REGION Network 44: E5CC[3]-Write TempSP + AlarmValue1 ~ AlarmValue2_LowerLimit Command
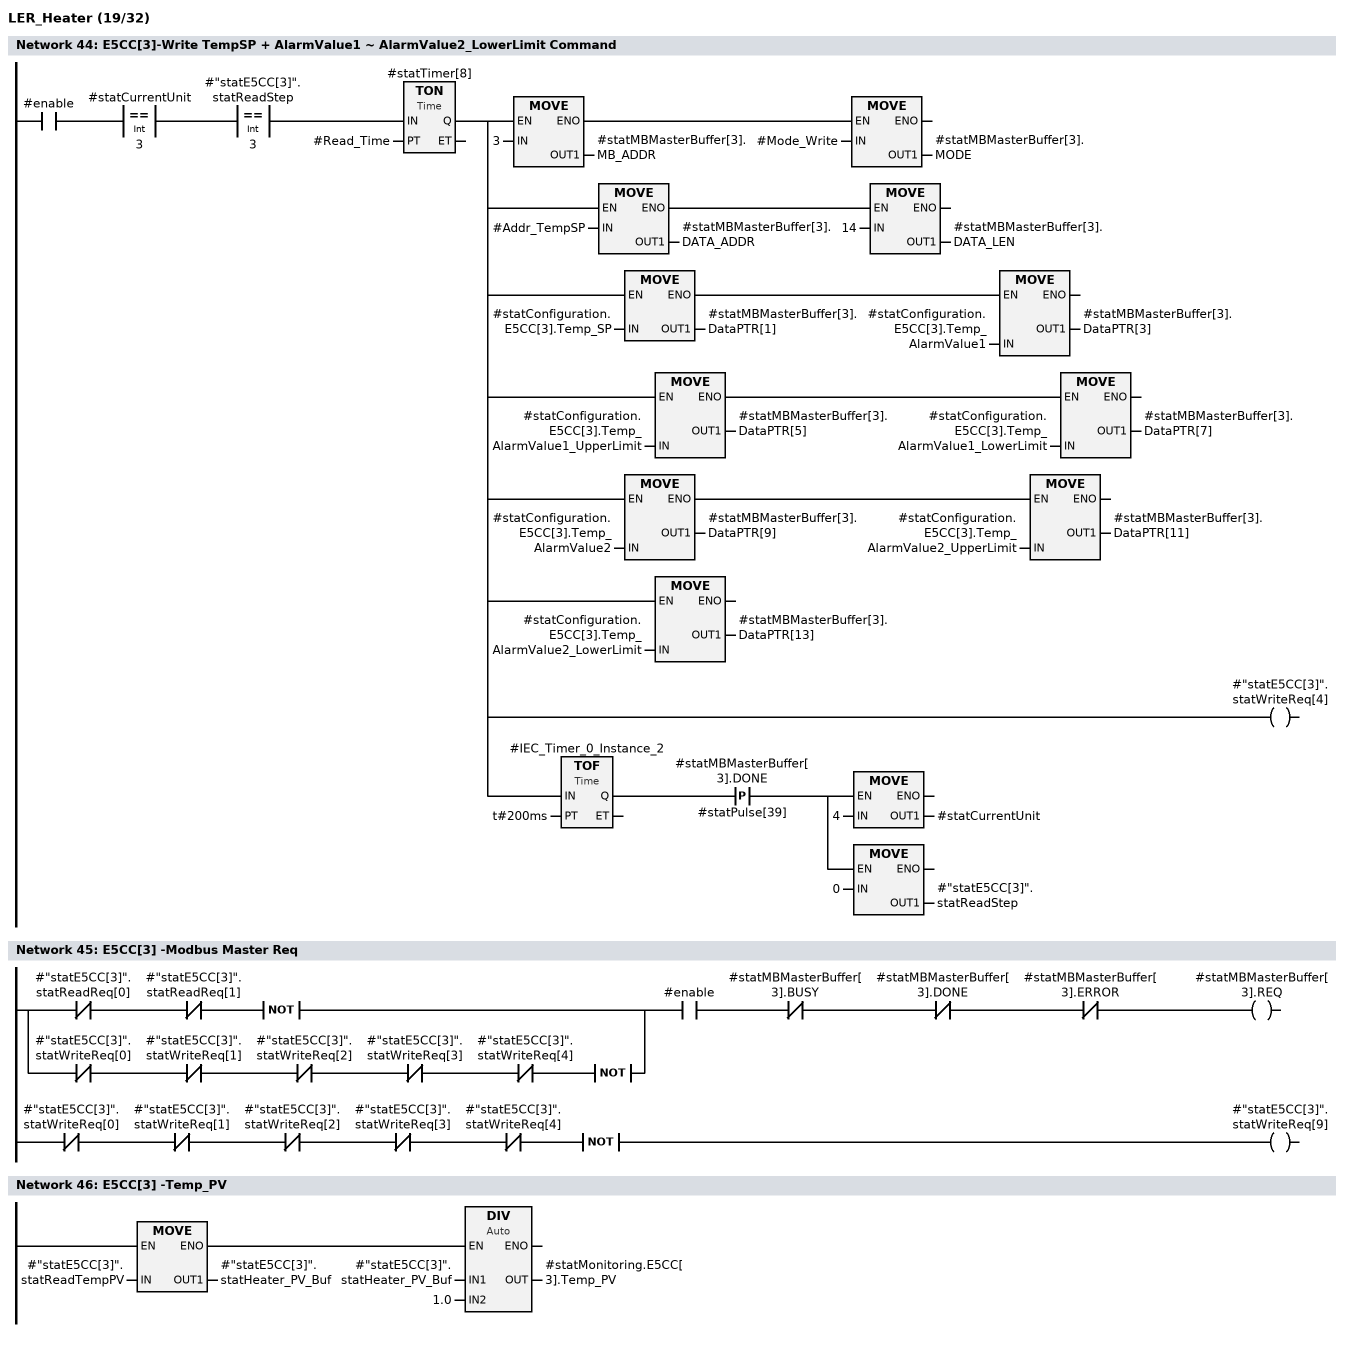
   RUNG wire#powerrail
      Contact( #enable )
      { S7_Templates := "SrcType := Int" } EQ_Contact(in1 := #statCurrentUnit, in2 := 3)
      { S7_Templates := "SrcType := Int" } EQ_Contact(in1 := #"statE5CC[3]".statReadStep, in2 := 3)
      { S7_Templates := "time_type := Time" } #statTimer[8].TON(pt := #Read_Time, et =>)
      wire#w1
      Move(in := 3, out1 => #statMBMasterBuffer[3].MB_ADDR)
      Move(in := #Mode_Write, out1 => #statMBMasterBuffer[3].MODE)
   END_RUNG
   RUNG wire#w1
      Move(in := #Addr_TempSP, out1 => #statMBMasterBuffer[3].DATA_ADDR)
      Move(in := 14, out1 => #statMBMasterBuffer[3].DATA_LEN)
   END_RUNG
   RUNG wire#w1
      Move(in := #statConfiguration.E5CC[3].Temp_SP, out1 => #statMBMasterBuffer[3].DataPTR[1])
      Move(in := #statConfiguration.E5CC[3].Temp_AlarmValue1, out1 => #statMBMasterBuffer[3].DataPTR[3])
   END_RUNG
   RUNG wire#w1
      Move(in := #statConfiguration.E5CC[3].Temp_AlarmValue1_UpperLimit, out1 => #statMBMasterBuffer[3].DataPTR[5])
      Move(in := #statConfiguration.E5CC[3].Temp_AlarmValue1_LowerLimit, out1 => #statMBMasterBuffer[3].DataPTR[7])
   END_RUNG
   RUNG wire#w1
      Move(in := #statConfiguration.E5CC[3].Temp_AlarmValue2, out1 => #statMBMasterBuffer[3].DataPTR[9])
      Move(in := #statConfiguration.E5CC[3].Temp_AlarmValue2_UpperLimit, out1 => #statMBMasterBuffer[3].DataPTR[11])
   END_RUNG
   RUNG wire#w1
      Move(in := #statConfiguration.E5CC[3].Temp_AlarmValue2_LowerLimit, out1 => #statMBMasterBuffer[3].DataPTR[13])
   END_RUNG
   RUNG wire#w1
      Coil( #"statE5CC[3]".statWriteReq[4] )
   END_RUNG
   RUNG wire#w1
      { S7_Templates := "time_type := Time" } #IEC_Timer_0_Instance_2.TOF(pt := t#200ms, et =>)
      P_Contact(operand := #statMBMasterBuffer[3].DONE, bit := #statPulse[39])
      wire#w2
      Move(in := 4, out1 => #statCurrentUnit)
   END_RUNG
   RUNG wire#w2
      Move(in := 0, out1 => #"statE5CC[3]".statReadStep)
   END_RUNG
   // the same network as SCL:
   #statTimer[8].TON(IN := #enable AND (#statCurrentUnit = 3) AND (#"statE5CC[3]".statReadStep = 3),
                     PT := #Read_Time);
   IF #statTimer[8].Q THEN
       #statMBMasterBuffer[3].MB_ADDR := 3;
       #statMBMasterBuffer[3].MODE := #Mode_Write;
       #statMBMasterBuffer[3].DATA_ADDR := #Addr_TempSP;
       #statMBMasterBuffer[3].DATA_LEN := 14;
       #statMBMasterBuffer[3].DataPTR[1] := #statConfiguration.E5CC[3].Temp_SP;
       #statMBMasterBuffer[3].DataPTR[3] := #statConfiguration.E5CC[3].Temp_AlarmValue1;
       #statMBMasterBuffer[3].DataPTR[5] := #statConfiguration.E5CC[3].Temp_AlarmValue1_UpperLimit;
       #statMBMasterBuffer[3].DataPTR[7] := #statConfiguration.E5CC[3].Temp_AlarmValue1_LowerLimit;
       #statMBMasterBuffer[3].DataPTR[9] := #statConfiguration.E5CC[3].Temp_AlarmValue2;
       #statMBMasterBuffer[3].DataPTR[11] := #statConfiguration.E5CC[3].Temp_AlarmValue2_UpperLimit;
       #statMBMasterBuffer[3].DataPTR[13] := #statConfiguration.E5CC[3].Temp_AlarmValue2_LowerLimit;
   END_IF;
   #"statE5CC[3]".statWriteReq[4] := #statTimer[8].Q;
   #IEC_Timer_0_Instance_2(IN := #statTimer[8].Q, PT := t#200ms);   // TOF
   #_w1 := #IEC_Timer_0_Instance_2.Q AND #statMBMasterBuffer[3].DONE AND NOT #statPulse[39];   // rising edge of #statMBMasterBuffer[3].DONE
   #statPulse[39] := #statMBMasterBuffer[3].DONE;
   IF #_w1 THEN
       #statCurrentUnit := 4;
       #"statE5CC[3]".statReadStep := 0;
   END_IF;
END_REGION

REGION Network 45: E5CC[3] -Modbus Master Req
   RUNG wire#powerrail
      I_Contact( #"statE5CC[3]".statReadReq[0] )
      I_Contact( #"statE5CC[3]".statReadReq[1] )
      Not()
      wire#w1
      Contact( #enable )
      I_Contact( #statMBMasterBuffer[3].BUSY )
      I_Contact( #statMBMasterBuffer[3].DONE )
      I_Contact( #statMBMasterBuffer[3].ERROR )
      Coil( #statMBMasterBuffer[3].REQ )
   END_RUNG
   RUNG wire#powerrail
      I_Contact( #"statE5CC[3]".statWriteReq[0] )
      I_Contact( #"statE5CC[3]".statWriteReq[1] )
      I_Contact( #"statE5CC[3]".statWriteReq[2] )
      I_Contact( #"statE5CC[3]".statWriteReq[3] )
      I_Contact( #"statE5CC[3]".statWriteReq[4] )
      Not()
   END_RUNG wire#w1
   RUNG wire#powerrail
      I_Contact( #"statE5CC[3]".statWriteReq[0] )
      I_Contact( #"statE5CC[3]".statWriteReq[1] )
      I_Contact( #"statE5CC[3]".statWriteReq[2] )
      I_Contact( #"statE5CC[3]".statWriteReq[3] )
      I_Contact( #"statE5CC[3]".statWriteReq[4] )
      Not()
      Coil( #"statE5CC[3]".statWriteReq[9] )
   END_RUNG
   // the same network as SCL:
   #statMBMasterBuffer[3].REQ := (NOT (NOT #"statE5CC[3]".statReadReq[0] AND NOT #"statE5CC[3]".statReadReq[1]) OR NOT (NOT #"statE5CC[3]".statWriteReq[0] AND NOT #"statE5CC[3]".statWriteReq[1] AND NOT #"statE5CC[3]".statWriteReq[2] AND NOT #"statE5CC[3]".statWriteReq[3] AND NOT #"statE5CC[3]".statWriteReq[4])) AND #enable AND NOT #statMBMasterBuffer[3].BUSY AND NOT #statMBMasterBuffer[3].DONE AND NOT #statMBMasterBuffer[3].ERROR;
   #"statE5CC[3]".statWriteReq[9] := NOT (NOT #"statE5CC[3]".statWriteReq[0] AND NOT #"statE5CC[3]".statWriteReq[1] AND NOT #"statE5CC[3]".statWriteReq[2] AND NOT #"statE5CC[3]".statWriteReq[3] AND NOT #"statE5CC[3]".statWriteReq[4]);
END_REGION

REGION Network 46: E5CC[3] -Temp_PV
   RUNG wire#powerrail
      Move(in := #"statE5CC[3]".statReadTempPV, out1 => #"statE5CC[3]".statHeater_PV_Buf)
      Div(in1 := #"statE5CC[3]".statHeater_PV_Buf, in2 := 1.0, out => #statMonitoring.E5CC[3].Temp_PV)
   END_RUNG
   // the same network as SCL:
   #"statE5CC[3]".statHeater_PV_Buf := #"statE5CC[3]".statReadTempPV;
   #statMonitoring.E5CC[3].Temp_PV := #"statE5CC[3]".statHeater_PV_Buf / 1.0;
END_REGION

REGION Network 47: E5CC[3] -Temp_PV Complete Check
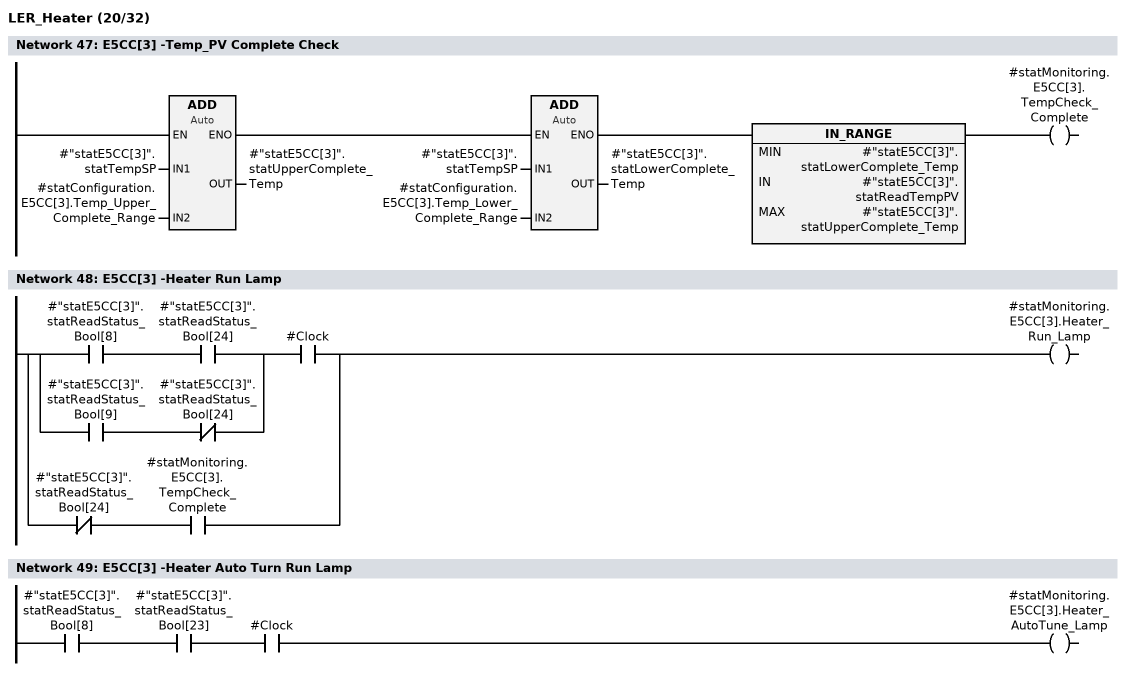
   RUNG wire#powerrail
      Add(in1 := #"statE5CC[3]".statTempSP, in2 := #statConfiguration.E5CC[3].Temp_Upper_Complete_Range, out => #"statE5CC[3]".statUpperComplete_Temp)
      Add(in1 := #"statE5CC[3]".statTempSP, in2 := #statConfiguration.E5CC[3].Temp_Lower_Complete_Range, out => #"statE5CC[3]".statLowerComplete_Temp)
      { S7_Templates := "SrcType := Real" } InRange(min := #"statE5CC[3]".statLowerComplete_Temp, in := #"statE5CC[3]".statReadTempPV, max := #"statE5CC[3]".statUpperComplete_Temp)
      Coil( #statMonitoring.E5CC[3].TempCheck_Complete )
   END_RUNG
   // the same network as SCL:
   #"statE5CC[3]".statUpperComplete_Temp := #"statE5CC[3]".statTempSP + #statConfiguration.E5CC[3].Temp_Upper_Complete_Range;
   #"statE5CC[3]".statLowerComplete_Temp := #"statE5CC[3]".statTempSP + #statConfiguration.E5CC[3].Temp_Lower_Complete_Range;
   #statMonitoring.E5CC[3].TempCheck_Complete := (#"statE5CC[3]".statLowerComplete_Temp <= #"statE5CC[3]".statReadTempPV) AND (#"statE5CC[3]".statReadTempPV <= #"statE5CC[3]".statUpperComplete_Temp);
END_REGION

REGION Network 48: E5CC[3] -Heater Run Lamp
   RUNG wire#powerrail
      Contact( #"statE5CC[3]".statReadStatus_Bool[8] )
      Contact( #"statE5CC[3]".statReadStatus_Bool[24] )
      wire#w1
      Contact( #Clock )
      wire#w2
      Coil( #statMonitoring.E5CC[3].Heater_Run_Lamp )
   END_RUNG
   RUNG wire#powerrail
      Contact( #"statE5CC[3]".statReadStatus_Bool[9] )
      I_Contact( #"statE5CC[3]".statReadStatus_Bool[24] )
   END_RUNG wire#w1
   RUNG wire#powerrail
      I_Contact( #"statE5CC[3]".statReadStatus_Bool[24] )
      Contact( #statMonitoring.E5CC[3].TempCheck_Complete )
   END_RUNG wire#w2
   // the same network as SCL:
   #statMonitoring.E5CC[3].Heater_Run_Lamp := (((#"statE5CC[3]".statReadStatus_Bool[8] AND #"statE5CC[3]".statReadStatus_Bool[24]) OR (#"statE5CC[3]".statReadStatus_Bool[9] AND NOT #"statE5CC[3]".statReadStatus_Bool[24])) AND #Clock) OR (NOT #"statE5CC[3]".statReadStatus_Bool[24] AND #statMonitoring.E5CC[3].TempCheck_Complete);
END_REGION

REGION Network 49: E5CC[3] -Heater Auto Turn Run Lamp
   RUNG wire#powerrail
      Contact( #"statE5CC[3]".statReadStatus_Bool[8] )
      Contact( #"statE5CC[3]".statReadStatus_Bool[23] )
      Contact( #Clock )
      Coil( #statMonitoring.E5CC[3].Heater_AutoTune_Lamp )
   END_RUNG
   // the same network as SCL:
   #statMonitoring.E5CC[3].Heater_AutoTune_Lamp := #"statE5CC[3]".statReadStatus_Bool[8] AND #"statE5CC[3]".statReadStatus_Bool[23] AND #Clock;
END_REGION

REGION Network 50 (SCL): E5CC[3] -Error Check
   REGION  E5CC Error Status
       // Dword to Bool
       SCATTER(IN := #"statE5CC[3]".statReadStatus,
               OUT => #"statE5CC[3]".statReadStatus_Bool);
   END_REGION


   REGION Error Code Search
       IF #"statE5CC[3]".statReadStatus <> 0 THEN
           CASE #"statE5CC[3]".statReadStatus OF
               #ERR_HEATER_CURRENT_VALUE_EXCEEDED_CT1:
                   #statMonitoring.E5CC[3].Status := #ERR_HEATER_CURRENT_VALUE_EXCEEDED_CT1;
               #ERR_HEATER_CURRENT_VALUE_HOLD_CT1:
                   #statMonitoring.E5CC[3].Status := #ERR_HEATER_CURRENT_VALUE_HOLD_CT1;
               #ERR_AD_CONVERTER_ABNORMALITY:
                   #statMonitoring.E5CC[3].Status := #ERR_AD_CONVERTER_ABNORMALITY;
               #ERR_HS_SSR_FAULT_ALERT_CT1:
                   #statMonitoring.E5CC[3].Status := #ERR_HS_SSR_FAULT_ALERT_CT1;
               #ERR_RSP_INPUT_ABNORMALITIES:
                   #statMonitoring.E5CC[3].Status := #ERR_RSP_INPUT_ABNORMALITIES;
               #ERR_MORE_THAN_INPUT:
                   #statMonitoring.E5CC[3].Status := #ERR_MORE_THAN_INPUT;
               #ERR_POTENTIOMETER_INPUT_ABNORMAL:
                   #statMonitoring.E5CC[3].Status := #ERR_POTENTIOMETER_INPUT_ABNORMAL;
               #ERR_CONTROL_OUTPUT_HEATED_OPEN_OUTPUT:
                   #statMonitoring.E5CC[3].Status := #ERR_CONTROL_OUTPUT_HEATED_OPEN_OUTPUT;
               #ERR_CONTROL_OUTPUT_COOL_CLOSE_OUTPUT:
                   #statMonitoring.E5CC[3].Status := #ERR_CONTROL_OUTPUT_COOL_CLOSE_OUTPUT;
               #ERR_HEATER_OPEN_CIRCUIT_HB_ALARM_CT1:
                   #statMonitoring.E5CC[3].Status := #ERR_HEATER_OPEN_CIRCUIT_HB_ALARM_CT1;
               #ERR_HEATER_OPEN_CIRCUIT_HB_ALARM_CT2:
                   #statMonitoring.E5CC[3].Status := #ERR_HEATER_OPEN_CIRCUIT_HB_ALARM_CT2;
               #ERR_ALERT_1:
                   #statMonitoring.E5CC[3].Status := #ERR_ALERT_1;
               #ERR_ALERT_2:
                   #statMonitoring.E5CC[3].Status := #ERR_ALERT_2;
               #ERR_ALERT_3:
                   #statMonitoring.E5CC[3].Status := #ERR_ALERT_3;
               #ERR_PROGRAM_END_OUTPUT:
                   #statMonitoring.E5CC[3].Status := #ERR_PROGRAM_END_OUTPUT;
               #ERR_EVENT_INPUT_1:
                   #statMonitoring.E5CC[3].Status := #ERR_EVENT_INPUT_1;
               #ERR_EVENT_INPUT_2:
                   #statMonitoring.E5CC[3].Status := #ERR_EVENT_INPUT_2;
               #ERR_EVENT_INPUT_3:
                   #statMonitoring.E5CC[3].Status := #ERR_EVENT_INPUT_3;
               #ERR_EVENT_INPUT_4:
                   #statMonitoring.E5CC[3].Status := #ERR_EVENT_INPUT_4;
               #ERR_WRITE_MODE:
                   #statMonitoring.E5CC[3].Status := #ERR_WRITE_MODE;
               #ERR_NON_VOLATILE_MEMORY:
                   #statMonitoring.E5CC[3].Status := #ERR_NON_VOLATILE_MEMORY;
               #ERR_SETTING_AREA:
                   #statMonitoring.E5CC[3].Status := #ERR_SETTING_AREA;
               #ERR_AT_RUN_STOP:
                   #statMonitoring.E5CC[3].Status := #ERR_AT_RUN_STOP;
               #ERR_RUN_STOP:
                   #statMonitoring.E5CC[3].Status := #ERR_RUN_STOP;
               #ERR_COMMUNICATION_WRITE:
                   #statMonitoring.E5CC[3].Status := #ERR_COMMUNICATION_WRITE;
               #ERR_AUTO_MANUAL:
                   #statMonitoring.E5CC[3].Status := #ERR_AUTO_MANUAL;
               #ERR_PROGRAM_START:
                   #statMonitoring.E5CC[3].Status := #ERR_PROGRAM_START;
               #ERR_HEATER_CURRENT_VALUE_EXCEEDED_CT2:
                   #statMonitoring.E5CC[3].Status := #ERR_HEATER_CURRENT_VALUE_EXCEEDED_CT2;
               #ERR_HEATER_CURRENT_VALUE_HOLD_CT2:
                   #statMonitoring.E5CC[3].Status := #ERR_HEATER_CURRENT_VALUE_HOLD_CT2;
               #ERR_HS_SSR_FAILURE_ALARM_CT2:
                   #statMonitoring.E5CC[3].Status := #ERR_HS_SSR_FAILURE_ALARM_CT2;
           END_CASE;
       ELSIF #"statE5CC[3]".statReadStatus = 0 THEN
           #statMonitoring.E5CC[3].Status := 0;
       END_IF;
   END_REGION

   #statMonitoring.E5CC[3].Error := #"statE5CC[3]".statReadStatus <> 0;
END_REGION

REGION Network 51 (SCL): E5CC[3]-##### Outputs mapping #####
   // Output Mapping
   #statMonitoring.E5CC[3].Temp_SP := #"statE5CC[3]".statTempSP;
   #statMonitoring.E5CC[3].Temp_AlarmValue1 := #"statE5CC[3]".statAlarmValue1;
   #statMonitoring.E5CC[3].Temp_AlarmValue1_UpperLimit := #"statE5CC[3]".statAlarmValue1_UpperLimit;
   #statMonitoring.E5CC[3].Temp_AlarmValue1_LowerLimit := #"statE5CC[3]".statAlarmValue1_LowerLimit;
   #statMonitoring.E5CC[3].Temp_AlarmValue2 := #"statE5CC[3]".statAlarmValue2;
   #statMonitoring.E5CC[3].Temp_AlarmValue2_UpperLimit := #"statE5CC[3]".statAlarmValue2_UpperLimit;
   #statMonitoring.E5CC[3].Temp_AlarmValue2_LowerLimit := #"statE5CC[3]".statAlarmValue2_LowerLimit;
   #statMonitoring.E5CC[3].E5CC_Status := #"statE5CC[3]".statReadStatus;
   #statMonitoring.E5CC[3].E5CC_Status_Bool := #"statE5CC[3]".statReadStatus_Bool;
END_REGION

REGION Network 52: E5CC[4] - ###### Input Mapping ######
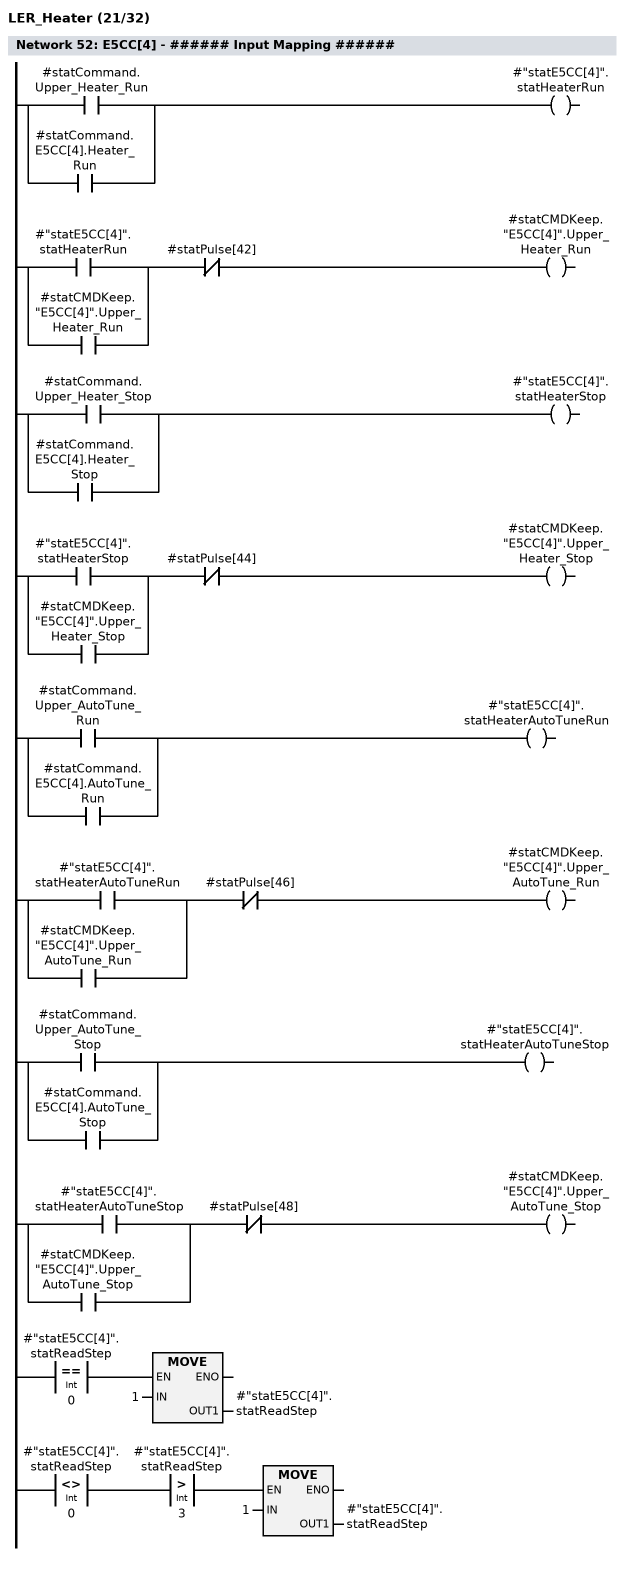
   RUNG wire#powerrail
      Contact( #statCommand.Upper_Heater_Run )
      wire#w1
      Coil( #"statE5CC[4]".statHeaterRun )
   END_RUNG
   RUNG wire#powerrail
      Contact( #statCommand.E5CC[4].Heater_Run )
   END_RUNG wire#w1
   RUNG wire#powerrail
      Contact( #"statE5CC[4]".statHeaterRun )
      wire#w2
      I_Contact( #statPulse[42] )
      Coil( #statCMDKeep."E5CC[4]".Upper_Heater_Run )
   END_RUNG
   RUNG wire#powerrail
      Contact( #statCMDKeep."E5CC[4]".Upper_Heater_Run )
   END_RUNG wire#w2
   RUNG wire#powerrail
      Contact( #statCommand.Upper_Heater_Stop )
      wire#w3
      Coil( #"statE5CC[4]".statHeaterStop )
   END_RUNG
   RUNG wire#powerrail
      Contact( #statCommand.E5CC[4].Heater_Stop )
   END_RUNG wire#w3
   RUNG wire#powerrail
      Contact( #"statE5CC[4]".statHeaterStop )
      wire#w4
      I_Contact( #statPulse[44] )
      Coil( #statCMDKeep."E5CC[4]".Upper_Heater_Stop )
   END_RUNG
   RUNG wire#powerrail
      Contact( #statCMDKeep."E5CC[4]".Upper_Heater_Stop )
   END_RUNG wire#w4
   RUNG wire#powerrail
      Contact( #statCommand.Upper_AutoTune_Run )
      wire#w5
      Coil( #"statE5CC[4]".statHeaterAutoTuneRun )
   END_RUNG
   RUNG wire#powerrail
      Contact( #statCommand.E5CC[4].AutoTune_Run )
   END_RUNG wire#w5
   RUNG wire#powerrail
      Contact( #"statE5CC[4]".statHeaterAutoTuneRun )
      wire#w6
      I_Contact( #statPulse[46] )
      Coil( #statCMDKeep."E5CC[4]".Upper_AutoTune_Run )
   END_RUNG
   RUNG wire#powerrail
      Contact( #statCMDKeep."E5CC[4]".Upper_AutoTune_Run )
   END_RUNG wire#w6
   RUNG wire#powerrail
      Contact( #statCommand.Upper_AutoTune_Stop )
      wire#w7
      Coil( #"statE5CC[4]".statHeaterAutoTuneStop )
   END_RUNG
   RUNG wire#powerrail
      Contact( #statCommand.E5CC[4].AutoTune_Stop )
   END_RUNG wire#w7
   RUNG wire#powerrail
      Contact( #"statE5CC[4]".statHeaterAutoTuneStop )
      wire#w8
      I_Contact( #statPulse[48] )
      Coil( #statCMDKeep."E5CC[4]".Upper_AutoTune_Stop )
   END_RUNG
   RUNG wire#powerrail
      Contact( #statCMDKeep."E5CC[4]".Upper_AutoTune_Stop )
   END_RUNG wire#w8
   RUNG wire#powerrail
      { S7_Templates := "SrcType := Int" } EQ_Contact(in1 := #"statE5CC[4]".statReadStep, in2 := 0)
      Move(in := 1, out1 => #"statE5CC[4]".statReadStep)
   END_RUNG
   RUNG wire#powerrail
      { S7_Templates := "SrcType := Int" } NE_Contact(in1 := #"statE5CC[4]".statReadStep, in2 := 0)
      { S7_Templates := "SrcType := Int" } GT_Contact(in1 := #"statE5CC[4]".statReadStep, in2 := 3)
      Move(in := 1, out1 => #"statE5CC[4]".statReadStep)
   END_RUNG
   // the same network as SCL:
   #"statE5CC[4]".statHeaterRun := #statCommand.Upper_Heater_Run OR #statCommand.E5CC[4].Heater_Run;
   #statCMDKeep."E5CC[4]".Upper_Heater_Run := (#"statE5CC[4]".statHeaterRun OR #statCMDKeep."E5CC[4]".Upper_Heater_Run) AND NOT #statPulse[42];
   #"statE5CC[4]".statHeaterStop := #statCommand.Upper_Heater_Stop OR #statCommand.E5CC[4].Heater_Stop;
   #statCMDKeep."E5CC[4]".Upper_Heater_Stop := (#"statE5CC[4]".statHeaterStop OR #statCMDKeep."E5CC[4]".Upper_Heater_Stop) AND NOT #statPulse[44];
   #"statE5CC[4]".statHeaterAutoTuneRun := #statCommand.Upper_AutoTune_Run OR #statCommand.E5CC[4].AutoTune_Run;
   #statCMDKeep."E5CC[4]".Upper_AutoTune_Run := (#"statE5CC[4]".statHeaterAutoTuneRun OR #statCMDKeep."E5CC[4]".Upper_AutoTune_Run) AND NOT #statPulse[46];
   #"statE5CC[4]".statHeaterAutoTuneStop := #statCommand.Upper_AutoTune_Stop OR #statCommand.E5CC[4].AutoTune_Stop;
   #statCMDKeep."E5CC[4]".Upper_AutoTune_Stop := (#"statE5CC[4]".statHeaterAutoTuneStop OR #statCMDKeep."E5CC[4]".Upper_AutoTune_Stop) AND NOT #statPulse[48];
   IF #"statE5CC[4]".statReadStep = 0 THEN #"statE5CC[4]".statReadStep := 1; END_IF;
   IF (#"statE5CC[4]".statReadStep <> 0) AND (#"statE5CC[4]".statReadStep > 3) THEN
       #"statE5CC[4]".statReadStep := 1;
   END_IF;
END_REGION

REGION Network 53: E5CC[4] -Read Temp PV + Status Command
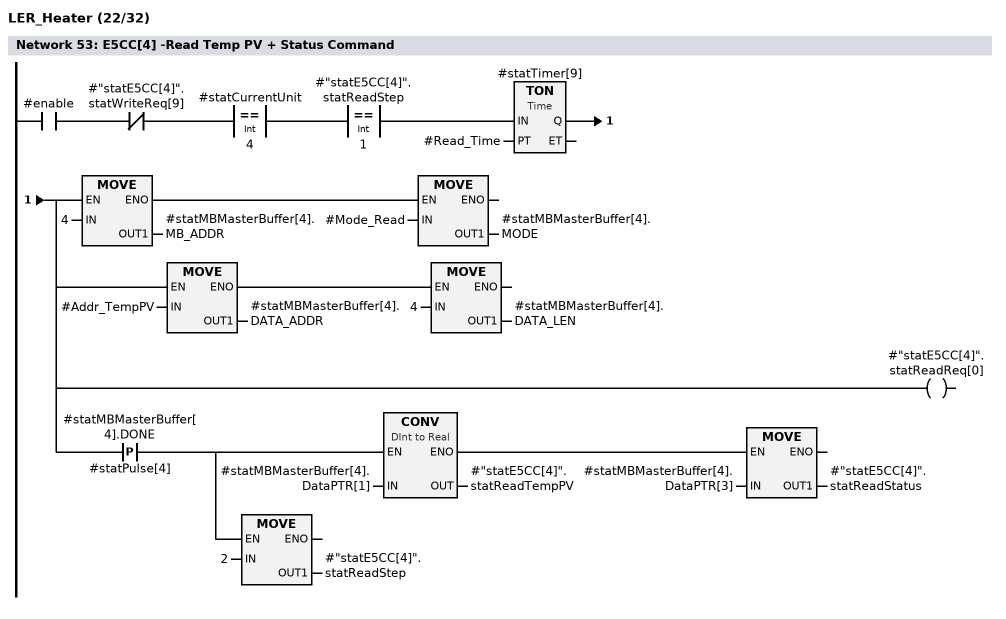
   RUNG wire#powerrail
      Contact( #enable )
      I_Contact( #"statE5CC[4]".statWriteReq[9] )
      { S7_Templates := "SrcType := Int" } EQ_Contact(in1 := #statCurrentUnit, in2 := 4)
      { S7_Templates := "SrcType := Int" } EQ_Contact(in1 := #"statE5CC[4]".statReadStep, in2 := 1)
      { S7_Templates := "time_type := Time" } #statTimer[9].TON(pt := #Read_Time, et =>)
      wire#w1
      Move(in := 4, out1 => #statMBMasterBuffer[4].MB_ADDR)
      Move(in := #Mode_Read, out1 => #statMBMasterBuffer[4].MODE)
   END_RUNG
   RUNG wire#w1
      Move(in := #Addr_TempPV, out1 => #statMBMasterBuffer[4].DATA_ADDR)
      Move(in := 4, out1 => #statMBMasterBuffer[4].DATA_LEN)
   END_RUNG
   RUNG wire#w1
      Coil( #"statE5CC[4]".statReadReq[0] )
   END_RUNG
   RUNG wire#w1
      P_Contact(operand := #statMBMasterBuffer[4].DONE, bit := #statPulse[4])
      wire#w2
      { S7_Templates := "[SrcType := DInt, DestType := Real]" } Convert(in := #statMBMasterBuffer[4].DataPTR[1], out => #"statE5CC[4]".statReadTempPV)
      Move(in := #statMBMasterBuffer[4].DataPTR[3], out1 => #"statE5CC[4]".statReadStatus)
   END_RUNG
   RUNG wire#w2
      Move(in := 2, out1 => #"statE5CC[4]".statReadStep)
   END_RUNG
   // the same network as SCL:
   #statTimer[9].TON(IN := #enable AND NOT #"statE5CC[4]".statWriteReq[9] AND (#statCurrentUnit = 4) AND (#"statE5CC[4]".statReadStep = 1),
                     PT := #Read_Time);
   IF #statTimer[9].Q THEN
       #statMBMasterBuffer[4].MB_ADDR := 4;
       #statMBMasterBuffer[4].MODE := #Mode_Read;
       #statMBMasterBuffer[4].DATA_ADDR := #Addr_TempPV;
       #statMBMasterBuffer[4].DATA_LEN := 4;
   END_IF;
   #"statE5CC[4]".statReadReq[0] := #statTimer[9].Q;
   #_w1 := #statTimer[9].Q AND #statMBMasterBuffer[4].DONE AND NOT #statPulse[4];   // rising edge of #statMBMasterBuffer[4].DONE
   #statPulse[4] := #statMBMasterBuffer[4].DONE;
   IF #_w1 THEN
       #"statE5CC[4]".statReadTempPV := DINT_TO_REAL(#statMBMasterBuffer[4].DataPTR[1]);
       #"statE5CC[4]".statReadStatus := #statMBMasterBuffer[4].DataPTR[3];
       #"statE5CC[4]".statReadStep := 2;
   END_IF;
END_REGION

REGION Network 54: E5CC[4] -Read TempSP + AlarmValue1 ~ AlarmValue2_LowerLimit Commad
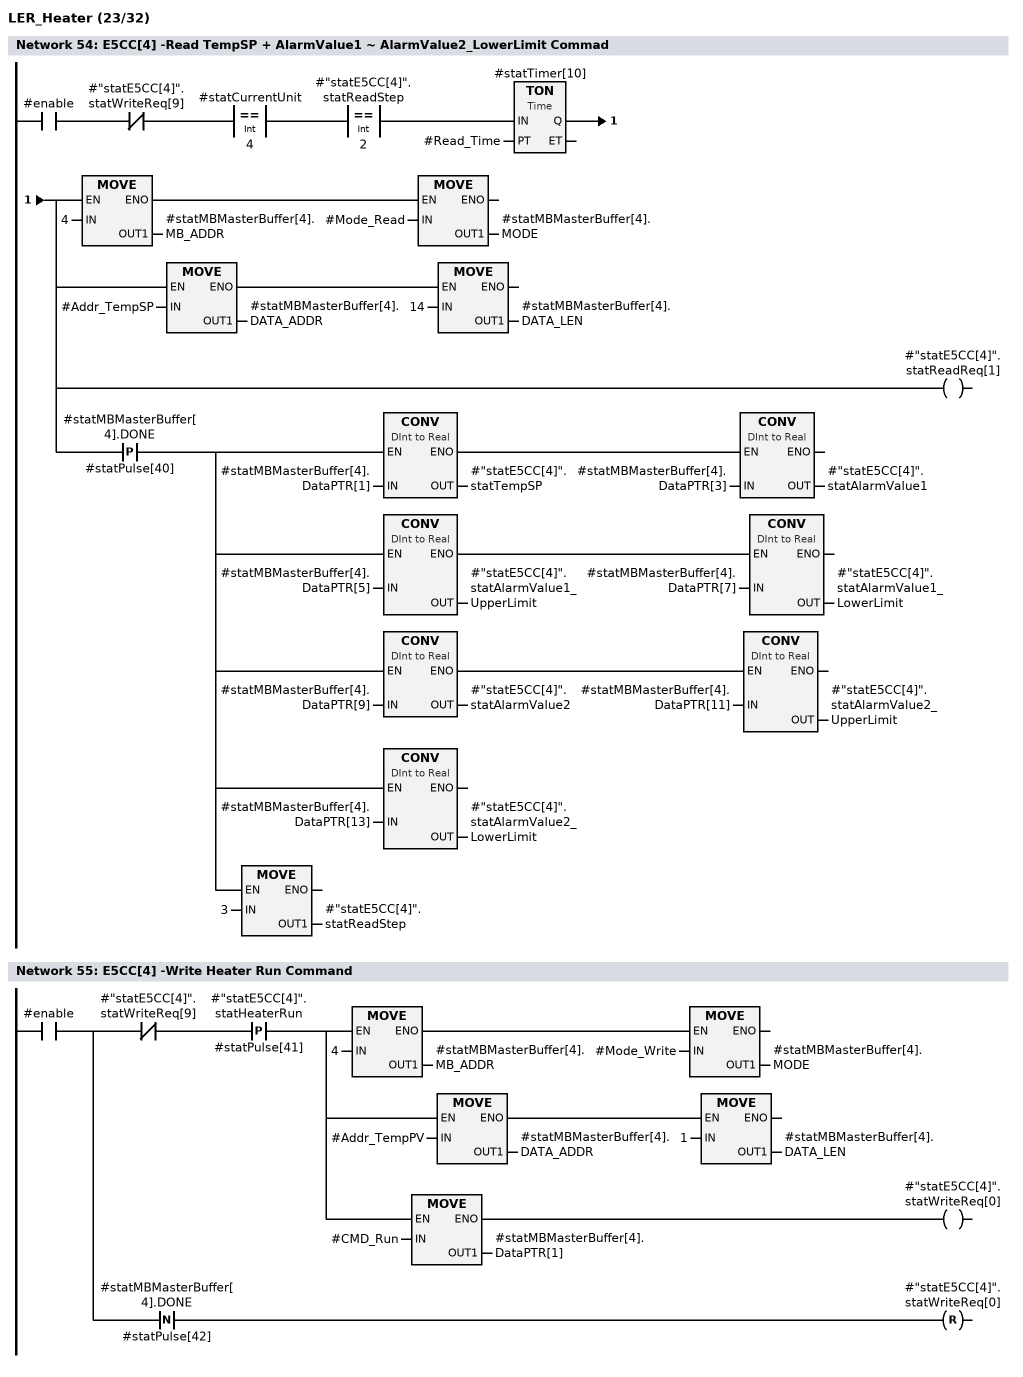
   RUNG wire#powerrail
      Contact( #enable )
      I_Contact( #"statE5CC[4]".statWriteReq[9] )
      { S7_Templates := "SrcType := Int" } EQ_Contact(in1 := #statCurrentUnit, in2 := 4)
      { S7_Templates := "SrcType := Int" } EQ_Contact(in1 := #"statE5CC[4]".statReadStep, in2 := 2)
      { S7_Templates := "time_type := Time" } #statTimer[10].TON(pt := #Read_Time, et =>)
      wire#w1
      Move(in := 4, out1 => #statMBMasterBuffer[4].MB_ADDR)
      Move(in := #Mode_Read, out1 => #statMBMasterBuffer[4].MODE)
   END_RUNG
   RUNG wire#w1
      Move(in := #Addr_TempSP, out1 => #statMBMasterBuffer[4].DATA_ADDR)
      Move(in := 14, out1 => #statMBMasterBuffer[4].DATA_LEN)
   END_RUNG
   RUNG wire#w1
      Coil( #"statE5CC[4]".statReadReq[1] )
   END_RUNG
   RUNG wire#w1
      P_Contact(operand := #statMBMasterBuffer[4].DONE, bit := #statPulse[40])
      wire#w2
      { S7_Templates := "[SrcType := DInt, DestType := Real]" } Convert(in := #statMBMasterBuffer[4].DataPTR[1], out => #"statE5CC[4]".statTempSP)
      { S7_Templates := "[SrcType := DInt, DestType := Real]" } Convert(in := #statMBMasterBuffer[4].DataPTR[3], out => #"statE5CC[4]".statAlarmValue1)
   END_RUNG
   RUNG wire#w2
      { S7_Templates := "[SrcType := DInt, DestType := Real]" } Convert(in := #statMBMasterBuffer[4].DataPTR[5], out => #"statE5CC[4]".statAlarmValue1_UpperLimit)
      { S7_Templates := "[SrcType := DInt, DestType := Real]" } Convert(in := #statMBMasterBuffer[4].DataPTR[7], out => #"statE5CC[4]".statAlarmValue1_LowerLimit)
   END_RUNG
   RUNG wire#w2
      { S7_Templates := "[SrcType := DInt, DestType := Real]" } Convert(in := #statMBMasterBuffer[4].DataPTR[9], out => #"statE5CC[4]".statAlarmValue2)
      { S7_Templates := "[SrcType := DInt, DestType := Real]" } Convert(in := #statMBMasterBuffer[4].DataPTR[11], out => #"statE5CC[4]".statAlarmValue2_UpperLimit)
   END_RUNG
   RUNG wire#w2
      { S7_Templates := "[SrcType := DInt, DestType := Real]" } Convert(in := #statMBMasterBuffer[4].DataPTR[13], out => #"statE5CC[4]".statAlarmValue2_LowerLimit)
   END_RUNG
   RUNG wire#w2
      Move(in := 3, out1 => #"statE5CC[4]".statReadStep)
   END_RUNG
   // the same network as SCL:
   #statTimer[10].TON(IN := #enable AND NOT #"statE5CC[4]".statWriteReq[9] AND (#statCurrentUnit = 4) AND (#"statE5CC[4]".statReadStep = 2),
                      PT := #Read_Time);
   IF #statTimer[10].Q THEN
       #statMBMasterBuffer[4].MB_ADDR := 4;
       #statMBMasterBuffer[4].MODE := #Mode_Read;
       #statMBMasterBuffer[4].DATA_ADDR := #Addr_TempSP;
       #statMBMasterBuffer[4].DATA_LEN := 14;
   END_IF;
   #"statE5CC[4]".statReadReq[1] := #statTimer[10].Q;
   #_w1 := #statTimer[10].Q AND #statMBMasterBuffer[4].DONE AND NOT #statPulse[40];   // rising edge of #statMBMasterBuffer[4].DONE
   #statPulse[40] := #statMBMasterBuffer[4].DONE;
   IF #_w1 THEN
       #"statE5CC[4]".statTempSP := DINT_TO_REAL(#statMBMasterBuffer[4].DataPTR[1]);
       #"statE5CC[4]".statAlarmValue1 := DINT_TO_REAL(#statMBMasterBuffer[4].DataPTR[3]);
       #"statE5CC[4]".statAlarmValue1_UpperLimit := DINT_TO_REAL(#statMBMasterBuffer[4].DataPTR[5]);
       #"statE5CC[4]".statAlarmValue1_LowerLimit := DINT_TO_REAL(#statMBMasterBuffer[4].DataPTR[7]);
       #"statE5CC[4]".statAlarmValue2 := DINT_TO_REAL(#statMBMasterBuffer[4].DataPTR[9]);
       #"statE5CC[4]".statAlarmValue2_UpperLimit := DINT_TO_REAL(#statMBMasterBuffer[4].DataPTR[11]);
       #"statE5CC[4]".statAlarmValue2_LowerLimit := DINT_TO_REAL(#statMBMasterBuffer[4].DataPTR[13]);
       #"statE5CC[4]".statReadStep := 3;
   END_IF;
END_REGION

REGION Network 55: E5CC[4] -Write Heater Run Command
   RUNG wire#powerrail
      Contact( #enable )
      wire#w1
      I_Contact( #"statE5CC[4]".statWriteReq[9] )
      P_Contact(operand := #"statE5CC[4]".statHeaterRun, bit := #statPulse[41])
      wire#w2
      Move(in := 4, out1 => #statMBMasterBuffer[4].MB_ADDR)
      Move(in := #Mode_Write, out1 => #statMBMasterBuffer[4].MODE)
   END_RUNG
   RUNG wire#w2
      Move(in := #Addr_TempPV, out1 => #statMBMasterBuffer[4].DATA_ADDR)
      Move(in := 1, out1 => #statMBMasterBuffer[4].DATA_LEN)
   END_RUNG
   RUNG wire#w2
      Move(in := #CMD_Run, out1 => #statMBMasterBuffer[4].DataPTR[1])
      Coil( #"statE5CC[4]".statWriteReq[0] )
   END_RUNG
   RUNG wire#w1
      N_Contact(operand := #statMBMasterBuffer[4].DONE, bit := #statPulse[42])
      R_Coil( #"statE5CC[4]".statWriteReq[0] )
   END_RUNG
   // the same network as SCL:
   #_w1 := #enable AND NOT #"statE5CC[4]".statWriteReq[9] AND #"statE5CC[4]".statHeaterRun AND NOT #statPulse[41];   // rising edge of #"statE5CC[4]".statHeaterRun
   #statPulse[41] := #"statE5CC[4]".statHeaterRun;
   IF #_w1 THEN
       #statMBMasterBuffer[4].MB_ADDR := 4;
       #statMBMasterBuffer[4].MODE := #Mode_Write;
       #statMBMasterBuffer[4].DATA_ADDR := #Addr_TempPV;
       #statMBMasterBuffer[4].DATA_LEN := 1;
       #statMBMasterBuffer[4].DataPTR[1] := #CMD_Run;
   END_IF;
   #"statE5CC[4]".statWriteReq[0] := #_w1;
   #_w2 := #enable AND NOT #statMBMasterBuffer[4].DONE AND #statPulse[42];   // falling edge of #statMBMasterBuffer[4].DONE
   #statPulse[42] := #statMBMasterBuffer[4].DONE;
   IF #_w2 THEN #"statE5CC[4]".statWriteReq[0] := FALSE; END_IF;
END_REGION

REGION Network 56: E5CC[4] -Write Heater Stop Command
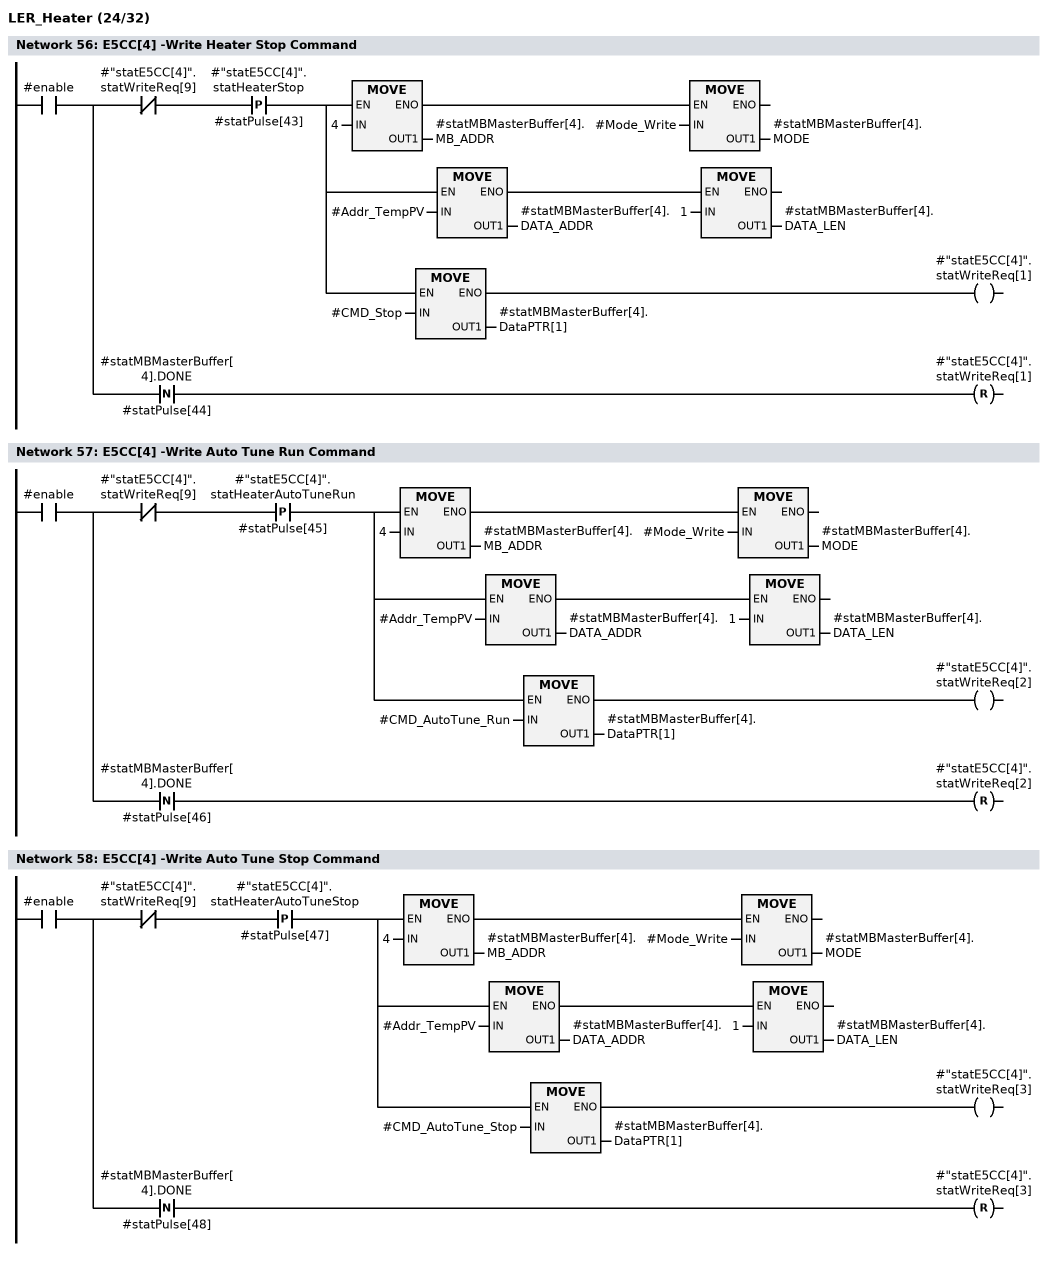
   RUNG wire#powerrail
      Contact( #enable )
      wire#w1
      I_Contact( #"statE5CC[4]".statWriteReq[9] )
      P_Contact(operand := #"statE5CC[4]".statHeaterStop, bit := #statPulse[43])
      wire#w2
      Move(in := 4, out1 => #statMBMasterBuffer[4].MB_ADDR)
      Move(in := #Mode_Write, out1 => #statMBMasterBuffer[4].MODE)
   END_RUNG
   RUNG wire#w2
      Move(in := #Addr_TempPV, out1 => #statMBMasterBuffer[4].DATA_ADDR)
      Move(in := 1, out1 => #statMBMasterBuffer[4].DATA_LEN)
   END_RUNG
   RUNG wire#w2
      Move(in := #CMD_Stop, out1 => #statMBMasterBuffer[4].DataPTR[1])
      Coil( #"statE5CC[4]".statWriteReq[1] )
   END_RUNG
   RUNG wire#w1
      N_Contact(operand := #statMBMasterBuffer[4].DONE, bit := #statPulse[44])
      R_Coil( #"statE5CC[4]".statWriteReq[1] )
   END_RUNG
   // the same network as SCL:
   #_w1 := #enable AND NOT #"statE5CC[4]".statWriteReq[9] AND #"statE5CC[4]".statHeaterStop AND NOT #statPulse[43];   // rising edge of #"statE5CC[4]".statHeaterStop
   #statPulse[43] := #"statE5CC[4]".statHeaterStop;
   IF #_w1 THEN
       #statMBMasterBuffer[4].MB_ADDR := 4;
       #statMBMasterBuffer[4].MODE := #Mode_Write;
       #statMBMasterBuffer[4].DATA_ADDR := #Addr_TempPV;
       #statMBMasterBuffer[4].DATA_LEN := 1;
       #statMBMasterBuffer[4].DataPTR[1] := #CMD_Stop;
   END_IF;
   #"statE5CC[4]".statWriteReq[1] := #_w1;
   #_w2 := #enable AND NOT #statMBMasterBuffer[4].DONE AND #statPulse[44];   // falling edge of #statMBMasterBuffer[4].DONE
   #statPulse[44] := #statMBMasterBuffer[4].DONE;
   IF #_w2 THEN #"statE5CC[4]".statWriteReq[1] := FALSE; END_IF;
END_REGION

REGION Network 57: E5CC[4] -Write Auto Tune Run Command
   RUNG wire#powerrail
      Contact( #enable )
      wire#w1
      I_Contact( #"statE5CC[4]".statWriteReq[9] )
      P_Contact(operand := #"statE5CC[4]".statHeaterAutoTuneRun, bit := #statPulse[45])
      wire#w2
      Move(in := 4, out1 => #statMBMasterBuffer[4].MB_ADDR)
      Move(in := #Mode_Write, out1 => #statMBMasterBuffer[4].MODE)
   END_RUNG
   RUNG wire#w2
      Move(in := #Addr_TempPV, out1 => #statMBMasterBuffer[4].DATA_ADDR)
      Move(in := 1, out1 => #statMBMasterBuffer[4].DATA_LEN)
   END_RUNG
   RUNG wire#w2
      Move(in := #CMD_AutoTune_Run, out1 => #statMBMasterBuffer[4].DataPTR[1])
      Coil( #"statE5CC[4]".statWriteReq[2] )
   END_RUNG
   RUNG wire#w1
      N_Contact(operand := #statMBMasterBuffer[4].DONE, bit := #statPulse[46])
      R_Coil( #"statE5CC[4]".statWriteReq[2] )
   END_RUNG
   // the same network as SCL:
   #_w1 := #enable AND NOT #"statE5CC[4]".statWriteReq[9] AND #"statE5CC[4]".statHeaterAutoTuneRun AND NOT #statPulse[45];   // rising edge of #"statE5CC[4]".statHeaterAutoTuneRun
   #statPulse[45] := #"statE5CC[4]".statHeaterAutoTuneRun;
   IF #_w1 THEN
       #statMBMasterBuffer[4].MB_ADDR := 4;
       #statMBMasterBuffer[4].MODE := #Mode_Write;
       #statMBMasterBuffer[4].DATA_ADDR := #Addr_TempPV;
       #statMBMasterBuffer[4].DATA_LEN := 1;
       #statMBMasterBuffer[4].DataPTR[1] := #CMD_AutoTune_Run;
   END_IF;
   #"statE5CC[4]".statWriteReq[2] := #_w1;
   #_w2 := #enable AND NOT #statMBMasterBuffer[4].DONE AND #statPulse[46];   // falling edge of #statMBMasterBuffer[4].DONE
   #statPulse[46] := #statMBMasterBuffer[4].DONE;
   IF #_w2 THEN #"statE5CC[4]".statWriteReq[2] := FALSE; END_IF;
END_REGION

REGION Network 58: E5CC[4] -Write Auto Tune Stop Command
   RUNG wire#powerrail
      Contact( #enable )
      wire#w1
      I_Contact( #"statE5CC[4]".statWriteReq[9] )
      P_Contact(operand := #"statE5CC[4]".statHeaterAutoTuneStop, bit := #statPulse[47])
      wire#w2
      Move(in := 4, out1 => #statMBMasterBuffer[4].MB_ADDR)
      Move(in := #Mode_Write, out1 => #statMBMasterBuffer[4].MODE)
   END_RUNG
   RUNG wire#w2
      Move(in := #Addr_TempPV, out1 => #statMBMasterBuffer[4].DATA_ADDR)
      Move(in := 1, out1 => #statMBMasterBuffer[4].DATA_LEN)
   END_RUNG
   RUNG wire#w2
      Move(in := #CMD_AutoTune_Stop, out1 => #statMBMasterBuffer[4].DataPTR[1])
      Coil( #"statE5CC[4]".statWriteReq[3] )
   END_RUNG
   RUNG wire#w1
      N_Contact(operand := #statMBMasterBuffer[4].DONE, bit := #statPulse[48])
      R_Coil( #"statE5CC[4]".statWriteReq[3] )
   END_RUNG
   // the same network as SCL:
   #_w1 := #enable AND NOT #"statE5CC[4]".statWriteReq[9] AND #"statE5CC[4]".statHeaterAutoTuneStop AND NOT #statPulse[47];   // rising edge of #"statE5CC[4]".statHeaterAutoTuneStop
   #statPulse[47] := #"statE5CC[4]".statHeaterAutoTuneStop;
   IF #_w1 THEN
       #statMBMasterBuffer[4].MB_ADDR := 4;
       #statMBMasterBuffer[4].MODE := #Mode_Write;
       #statMBMasterBuffer[4].DATA_ADDR := #Addr_TempPV;
       #statMBMasterBuffer[4].DATA_LEN := 1;
       #statMBMasterBuffer[4].DataPTR[1] := #CMD_AutoTune_Stop;
   END_IF;
   #"statE5CC[4]".statWriteReq[3] := #_w1;
   #_w2 := #enable AND NOT #statMBMasterBuffer[4].DONE AND #statPulse[48];   // falling edge of #statMBMasterBuffer[4].DONE
   #statPulse[48] := #statMBMasterBuffer[4].DONE;
   IF #_w2 THEN #"statE5CC[4]".statWriteReq[3] := FALSE; END_IF;
END_REGION

REGION Network 59: E5CC[4]-Write TempSP + AlarmValue1 ~ AlarmValue2_LowerLimit Command
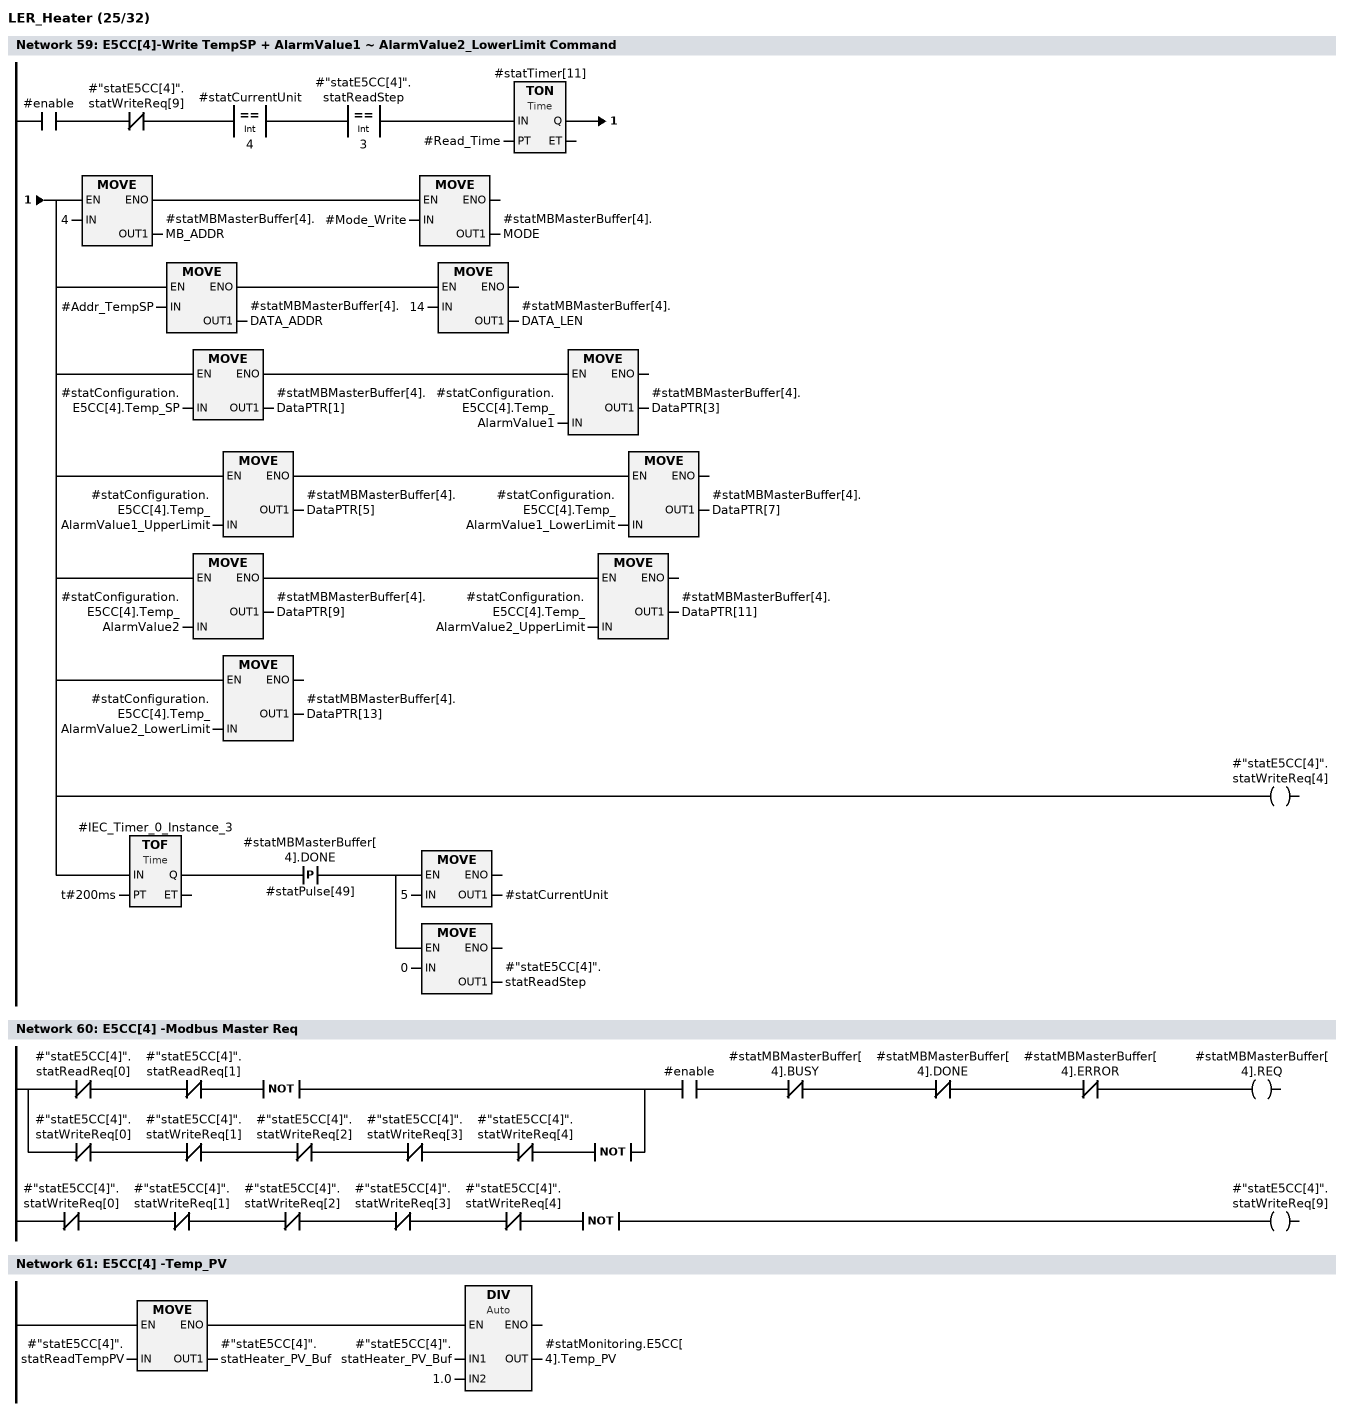
   RUNG wire#powerrail
      Contact( #enable )
      I_Contact( #"statE5CC[4]".statWriteReq[9] )
      { S7_Templates := "SrcType := Int" } EQ_Contact(in1 := #statCurrentUnit, in2 := 4)
      { S7_Templates := "SrcType := Int" } EQ_Contact(in1 := #"statE5CC[4]".statReadStep, in2 := 3)
      { S7_Templates := "time_type := Time" } #statTimer[11].TON(pt := #Read_Time, et =>)
      wire#w1
      Move(in := 4, out1 => #statMBMasterBuffer[4].MB_ADDR)
      Move(in := #Mode_Write, out1 => #statMBMasterBuffer[4].MODE)
   END_RUNG
   RUNG wire#w1
      Move(in := #Addr_TempSP, out1 => #statMBMasterBuffer[4].DATA_ADDR)
      Move(in := 14, out1 => #statMBMasterBuffer[4].DATA_LEN)
   END_RUNG
   RUNG wire#w1
      Move(in := #statConfiguration.E5CC[4].Temp_SP, out1 => #statMBMasterBuffer[4].DataPTR[1])
      Move(in := #statConfiguration.E5CC[4].Temp_AlarmValue1, out1 => #statMBMasterBuffer[4].DataPTR[3])
   END_RUNG
   RUNG wire#w1
      Move(in := #statConfiguration.E5CC[4].Temp_AlarmValue1_UpperLimit, out1 => #statMBMasterBuffer[4].DataPTR[5])
      Move(in := #statConfiguration.E5CC[4].Temp_AlarmValue1_LowerLimit, out1 => #statMBMasterBuffer[4].DataPTR[7])
   END_RUNG
   RUNG wire#w1
      Move(in := #statConfiguration.E5CC[4].Temp_AlarmValue2, out1 => #statMBMasterBuffer[4].DataPTR[9])
      Move(in := #statConfiguration.E5CC[4].Temp_AlarmValue2_UpperLimit, out1 => #statMBMasterBuffer[4].DataPTR[11])
   END_RUNG
   RUNG wire#w1
      Move(in := #statConfiguration.E5CC[4].Temp_AlarmValue2_LowerLimit, out1 => #statMBMasterBuffer[4].DataPTR[13])
   END_RUNG
   RUNG wire#w1
      Coil( #"statE5CC[4]".statWriteReq[4] )
   END_RUNG
   RUNG wire#w1
      { S7_Templates := "time_type := Time" } #IEC_Timer_0_Instance_3.TOF(pt := t#200ms, et =>)
      P_Contact(operand := #statMBMasterBuffer[4].DONE, bit := #statPulse[49])
      wire#w2
      Move(in := 5, out1 => #statCurrentUnit)
   END_RUNG
   RUNG wire#w2
      Move(in := 0, out1 => #"statE5CC[4]".statReadStep)
   END_RUNG
   // the same network as SCL:
   #statTimer[11].TON(IN := #enable AND NOT #"statE5CC[4]".statWriteReq[9] AND (#statCurrentUnit = 4) AND (#"statE5CC[4]".statReadStep = 3),
                      PT := #Read_Time);
   IF #statTimer[11].Q THEN
       #statMBMasterBuffer[4].MB_ADDR := 4;
       #statMBMasterBuffer[4].MODE := #Mode_Write;
       #statMBMasterBuffer[4].DATA_ADDR := #Addr_TempSP;
       #statMBMasterBuffer[4].DATA_LEN := 14;
       #statMBMasterBuffer[4].DataPTR[1] := #statConfiguration.E5CC[4].Temp_SP;
       #statMBMasterBuffer[4].DataPTR[3] := #statConfiguration.E5CC[4].Temp_AlarmValue1;
       #statMBMasterBuffer[4].DataPTR[5] := #statConfiguration.E5CC[4].Temp_AlarmValue1_UpperLimit;
       #statMBMasterBuffer[4].DataPTR[7] := #statConfiguration.E5CC[4].Temp_AlarmValue1_LowerLimit;
       #statMBMasterBuffer[4].DataPTR[9] := #statConfiguration.E5CC[4].Temp_AlarmValue2;
       #statMBMasterBuffer[4].DataPTR[11] := #statConfiguration.E5CC[4].Temp_AlarmValue2_UpperLimit;
       #statMBMasterBuffer[4].DataPTR[13] := #statConfiguration.E5CC[4].Temp_AlarmValue2_LowerLimit;
   END_IF;
   #"statE5CC[4]".statWriteReq[4] := #statTimer[11].Q;
   #IEC_Timer_0_Instance_3(IN := #statTimer[11].Q, PT := t#200ms);   // TOF
   #_w1 := #IEC_Timer_0_Instance_3.Q AND #statMBMasterBuffer[4].DONE AND NOT #statPulse[49];   // rising edge of #statMBMasterBuffer[4].DONE
   #statPulse[49] := #statMBMasterBuffer[4].DONE;
   IF #_w1 THEN
       #statCurrentUnit := 5;
       #"statE5CC[4]".statReadStep := 0;
   END_IF;
END_REGION

REGION Network 60: E5CC[4] -Modbus Master Req
   RUNG wire#powerrail
      I_Contact( #"statE5CC[4]".statReadReq[0] )
      I_Contact( #"statE5CC[4]".statReadReq[1] )
      Not()
      wire#w1
      Contact( #enable )
      I_Contact( #statMBMasterBuffer[4].BUSY )
      I_Contact( #statMBMasterBuffer[4].DONE )
      I_Contact( #statMBMasterBuffer[4].ERROR )
      Coil( #statMBMasterBuffer[4].REQ )
   END_RUNG
   RUNG wire#powerrail
      I_Contact( #"statE5CC[4]".statWriteReq[0] )
      I_Contact( #"statE5CC[4]".statWriteReq[1] )
      I_Contact( #"statE5CC[4]".statWriteReq[2] )
      I_Contact( #"statE5CC[4]".statWriteReq[3] )
      I_Contact( #"statE5CC[4]".statWriteReq[4] )
      Not()
   END_RUNG wire#w1
   RUNG wire#powerrail
      I_Contact( #"statE5CC[4]".statWriteReq[0] )
      I_Contact( #"statE5CC[4]".statWriteReq[1] )
      I_Contact( #"statE5CC[4]".statWriteReq[2] )
      I_Contact( #"statE5CC[4]".statWriteReq[3] )
      I_Contact( #"statE5CC[4]".statWriteReq[4] )
      Not()
      Coil( #"statE5CC[4]".statWriteReq[9] )
   END_RUNG
   // the same network as SCL:
   #statMBMasterBuffer[4].REQ := (NOT (NOT #"statE5CC[4]".statReadReq[0] AND NOT #"statE5CC[4]".statReadReq[1]) OR NOT (NOT #"statE5CC[4]".statWriteReq[0] AND NOT #"statE5CC[4]".statWriteReq[1] AND NOT #"statE5CC[4]".statWriteReq[2] AND NOT #"statE5CC[4]".statWriteReq[3] AND NOT #"statE5CC[4]".statWriteReq[4])) AND #enable AND NOT #statMBMasterBuffer[4].BUSY AND NOT #statMBMasterBuffer[4].DONE AND NOT #statMBMasterBuffer[4].ERROR;
   #"statE5CC[4]".statWriteReq[9] := NOT (NOT #"statE5CC[4]".statWriteReq[0] AND NOT #"statE5CC[4]".statWriteReq[1] AND NOT #"statE5CC[4]".statWriteReq[2] AND NOT #"statE5CC[4]".statWriteReq[3] AND NOT #"statE5CC[4]".statWriteReq[4]);
END_REGION

REGION Network 61: E5CC[4] -Temp_PV
   RUNG wire#powerrail
      Move(in := #"statE5CC[4]".statReadTempPV, out1 => #"statE5CC[4]".statHeater_PV_Buf)
      Div(in1 := #"statE5CC[4]".statHeater_PV_Buf, in2 := 1.0, out => #statMonitoring.E5CC[4].Temp_PV)
   END_RUNG
   // the same network as SCL:
   #"statE5CC[4]".statHeater_PV_Buf := #"statE5CC[4]".statReadTempPV;
   #statMonitoring.E5CC[4].Temp_PV := #"statE5CC[4]".statHeater_PV_Buf / 1.0;
END_REGION

REGION Network 62: E5CC[4] -Temp_PV Complete Check
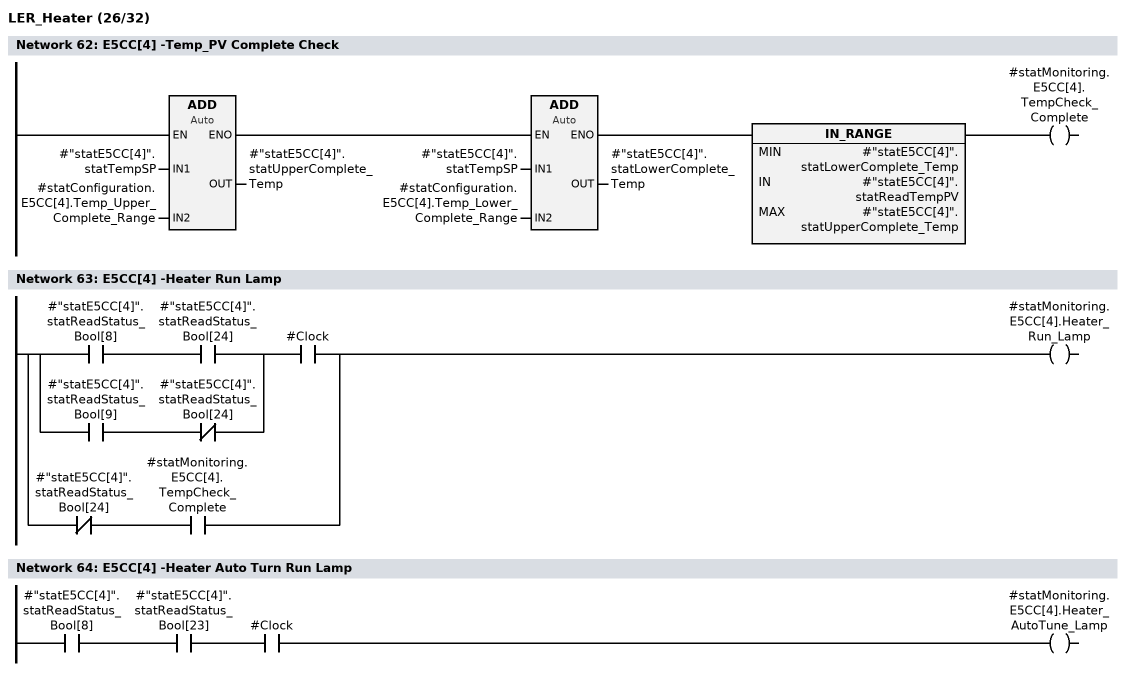
   RUNG wire#powerrail
      Add(in1 := #"statE5CC[4]".statTempSP, in2 := #statConfiguration.E5CC[4].Temp_Upper_Complete_Range, out => #"statE5CC[4]".statUpperComplete_Temp)
      Add(in1 := #"statE5CC[4]".statTempSP, in2 := #statConfiguration.E5CC[4].Temp_Lower_Complete_Range, out => #"statE5CC[4]".statLowerComplete_Temp)
      { S7_Templates := "SrcType := Real" } InRange(min := #"statE5CC[4]".statLowerComplete_Temp, in := #"statE5CC[4]".statReadTempPV, max := #"statE5CC[4]".statUpperComplete_Temp)
      Coil( #statMonitoring.E5CC[4].TempCheck_Complete )
   END_RUNG
   // the same network as SCL:
   #"statE5CC[4]".statUpperComplete_Temp := #"statE5CC[4]".statTempSP + #statConfiguration.E5CC[4].Temp_Upper_Complete_Range;
   #"statE5CC[4]".statLowerComplete_Temp := #"statE5CC[4]".statTempSP + #statConfiguration.E5CC[4].Temp_Lower_Complete_Range;
   #statMonitoring.E5CC[4].TempCheck_Complete := (#"statE5CC[4]".statLowerComplete_Temp <= #"statE5CC[4]".statReadTempPV) AND (#"statE5CC[4]".statReadTempPV <= #"statE5CC[4]".statUpperComplete_Temp);
END_REGION

REGION Network 63: E5CC[4] -Heater Run Lamp
   RUNG wire#powerrail
      Contact( #"statE5CC[4]".statReadStatus_Bool[8] )
      Contact( #"statE5CC[4]".statReadStatus_Bool[24] )
      wire#w1
      Contact( #Clock )
      wire#w2
      Coil( #statMonitoring.E5CC[4].Heater_Run_Lamp )
   END_RUNG
   RUNG wire#powerrail
      Contact( #"statE5CC[4]".statReadStatus_Bool[9] )
      I_Contact( #"statE5CC[4]".statReadStatus_Bool[24] )
   END_RUNG wire#w1
   RUNG wire#powerrail
      I_Contact( #"statE5CC[4]".statReadStatus_Bool[24] )
      Contact( #statMonitoring.E5CC[4].TempCheck_Complete )
   END_RUNG wire#w2
   // the same network as SCL:
   #statMonitoring.E5CC[4].Heater_Run_Lamp := (((#"statE5CC[4]".statReadStatus_Bool[8] AND #"statE5CC[4]".statReadStatus_Bool[24]) OR (#"statE5CC[4]".statReadStatus_Bool[9] AND NOT #"statE5CC[4]".statReadStatus_Bool[24])) AND #Clock) OR (NOT #"statE5CC[4]".statReadStatus_Bool[24] AND #statMonitoring.E5CC[4].TempCheck_Complete);
END_REGION

REGION Network 64: E5CC[4] -Heater Auto Turn Run Lamp
   RUNG wire#powerrail
      Contact( #"statE5CC[4]".statReadStatus_Bool[8] )
      Contact( #"statE5CC[4]".statReadStatus_Bool[23] )
      Contact( #Clock )
      Coil( #statMonitoring.E5CC[4].Heater_AutoTune_Lamp )
   END_RUNG
   // the same network as SCL:
   #statMonitoring.E5CC[4].Heater_AutoTune_Lamp := #"statE5CC[4]".statReadStatus_Bool[8] AND #"statE5CC[4]".statReadStatus_Bool[23] AND #Clock;
END_REGION

REGION Network 65 (SCL): E5CC[4] -Error Check
   REGION  E5CC Error Status
       // Dword to Bool
       SCATTER(IN := #"statE5CC[4]".statReadStatus,
               OUT => #"statE5CC[4]".statReadStatus_Bool);
   END_REGION


   REGION Error Code Search
       IF #"statE5CC[4]".statReadStatus <> 0 THEN
           CASE #"statE5CC[4]".statReadStatus OF
               #ERR_HEATER_CURRENT_VALUE_EXCEEDED_CT1:
                   #statMonitoring.E5CC[4].Status := #ERR_HEATER_CURRENT_VALUE_EXCEEDED_CT1;
               #ERR_HEATER_CURRENT_VALUE_HOLD_CT1:
                   #statMonitoring.E5CC[4].Status := #ERR_HEATER_CURRENT_VALUE_HOLD_CT1;
               #ERR_AD_CONVERTER_ABNORMALITY:
                   #statMonitoring.E5CC[4].Status := #ERR_AD_CONVERTER_ABNORMALITY;
               #ERR_HS_SSR_FAULT_ALERT_CT1:
                   #statMonitoring.E5CC[4].Status := #ERR_HS_SSR_FAULT_ALERT_CT1;
               #ERR_RSP_INPUT_ABNORMALITIES:
                   #statMonitoring.E5CC[4].Status := #ERR_RSP_INPUT_ABNORMALITIES;
               #ERR_MORE_THAN_INPUT:
                   #statMonitoring.E5CC[4].Status := #ERR_MORE_THAN_INPUT;
               #ERR_POTENTIOMETER_INPUT_ABNORMAL:
                   #statMonitoring.E5CC[4].Status := #ERR_POTENTIOMETER_INPUT_ABNORMAL;
               #ERR_CONTROL_OUTPUT_HEATED_OPEN_OUTPUT:
                   #statMonitoring.E5CC[4].Status := #ERR_CONTROL_OUTPUT_HEATED_OPEN_OUTPUT;
               #ERR_CONTROL_OUTPUT_COOL_CLOSE_OUTPUT:
                   #statMonitoring.E5CC[4].Status := #ERR_CONTROL_OUTPUT_COOL_CLOSE_OUTPUT;
               #ERR_HEATER_OPEN_CIRCUIT_HB_ALARM_CT1:
                   #statMonitoring.E5CC[4].Status := #ERR_HEATER_OPEN_CIRCUIT_HB_ALARM_CT1;
               #ERR_HEATER_OPEN_CIRCUIT_HB_ALARM_CT2:
                   #statMonitoring.E5CC[4].Status := #ERR_HEATER_OPEN_CIRCUIT_HB_ALARM_CT2;
               #ERR_ALERT_1:
                   #statMonitoring.E5CC[4].Status := #ERR_ALERT_1;
               #ERR_ALERT_2:
                   #statMonitoring.E5CC[4].Status := #ERR_ALERT_2;
               #ERR_ALERT_3:
                   #statMonitoring.E5CC[4].Status := #ERR_ALERT_3;
               #ERR_PROGRAM_END_OUTPUT:
                   #statMonitoring.E5CC[4].Status := #ERR_PROGRAM_END_OUTPUT;
               #ERR_EVENT_INPUT_1:
                   #statMonitoring.E5CC[4].Status := #ERR_EVENT_INPUT_1;
               #ERR_EVENT_INPUT_2:
                   #statMonitoring.E5CC[4].Status := #ERR_EVENT_INPUT_2;
               #ERR_EVENT_INPUT_3:
                   #statMonitoring.E5CC[4].Status := #ERR_EVENT_INPUT_3;
               #ERR_EVENT_INPUT_4:
                   #statMonitoring.E5CC[4].Status := #ERR_EVENT_INPUT_4;
               #ERR_WRITE_MODE:
                   #statMonitoring.E5CC[4].Status := #ERR_WRITE_MODE;
               #ERR_NON_VOLATILE_MEMORY:
                   #statMonitoring.E5CC[4].Status := #ERR_NON_VOLATILE_MEMORY;
               #ERR_SETTING_AREA:
                   #statMonitoring.E5CC[4].Status := #ERR_SETTING_AREA;
               #ERR_AT_RUN_STOP:
                   #statMonitoring.E5CC[4].Status := #ERR_AT_RUN_STOP;
               #ERR_RUN_STOP:
                   #statMonitoring.E5CC[4].Status := #ERR_RUN_STOP;
               #ERR_COMMUNICATION_WRITE:
                   #statMonitoring.E5CC[4].Status := #ERR_COMMUNICATION_WRITE;
               #ERR_AUTO_MANUAL:
                   #statMonitoring.E5CC[4].Status := #ERR_AUTO_MANUAL;
               #ERR_PROGRAM_START:
                   #statMonitoring.E5CC[4].Status := #ERR_PROGRAM_START;
               #ERR_HEATER_CURRENT_VALUE_EXCEEDED_CT2:
                   #statMonitoring.E5CC[4].Status := #ERR_HEATER_CURRENT_VALUE_EXCEEDED_CT2;
               #ERR_HEATER_CURRENT_VALUE_HOLD_CT2:
                   #statMonitoring.E5CC[4].Status := #ERR_HEATER_CURRENT_VALUE_HOLD_CT2;
               #ERR_HS_SSR_FAILURE_ALARM_CT2:
                   #statMonitoring.E5CC[4].Status := #ERR_HS_SSR_FAILURE_ALARM_CT2;
           END_CASE;
       ELSIF #"statE5CC[4]".statReadStatus = 0 THEN
           #statMonitoring.E5CC[4].Status := 0;
       END_IF;
   END_REGION

   #statMonitoring.E5CC[4].Error := #"statE5CC[4]".statReadStatus <> 0;
END_REGION

REGION Network 66 (SCL): E5CC[4]-##### Outputs mapping #####
   // Output Mapping
   #statMonitoring.E5CC[4].Temp_SP := #"statE5CC[4]".statTempSP;
   #statMonitoring.E5CC[4].Temp_AlarmValue1 := #"statE5CC[4]".statAlarmValue1;
   #statMonitoring.E5CC[4].Temp_AlarmValue1_UpperLimit := #"statE5CC[4]".statAlarmValue1_UpperLimit;
   #statMonitoring.E5CC[4].Temp_AlarmValue1_LowerLimit := #"statE5CC[4]".statAlarmValue1_LowerLimit;
   #statMonitoring.E5CC[4].Temp_AlarmValue2 := #"statE5CC[4]".statAlarmValue2;
   #statMonitoring.E5CC[4].Temp_AlarmValue2_UpperLimit := #"statE5CC[4]".statAlarmValue2_UpperLimit;
   #statMonitoring.E5CC[4].Temp_AlarmValue2_LowerLimit := #"statE5CC[4]".statAlarmValue2_LowerLimit;
   #statMonitoring.E5CC[4].E5CC_Status := #"statE5CC[4]".statReadStatus;
   #statMonitoring.E5CC[4].E5CC_Status_Bool := #"statE5CC[4]".statReadStatus_Bool;
END_REGION

REGION Network 67: E5CC[5] - ###### Input Mapping ######
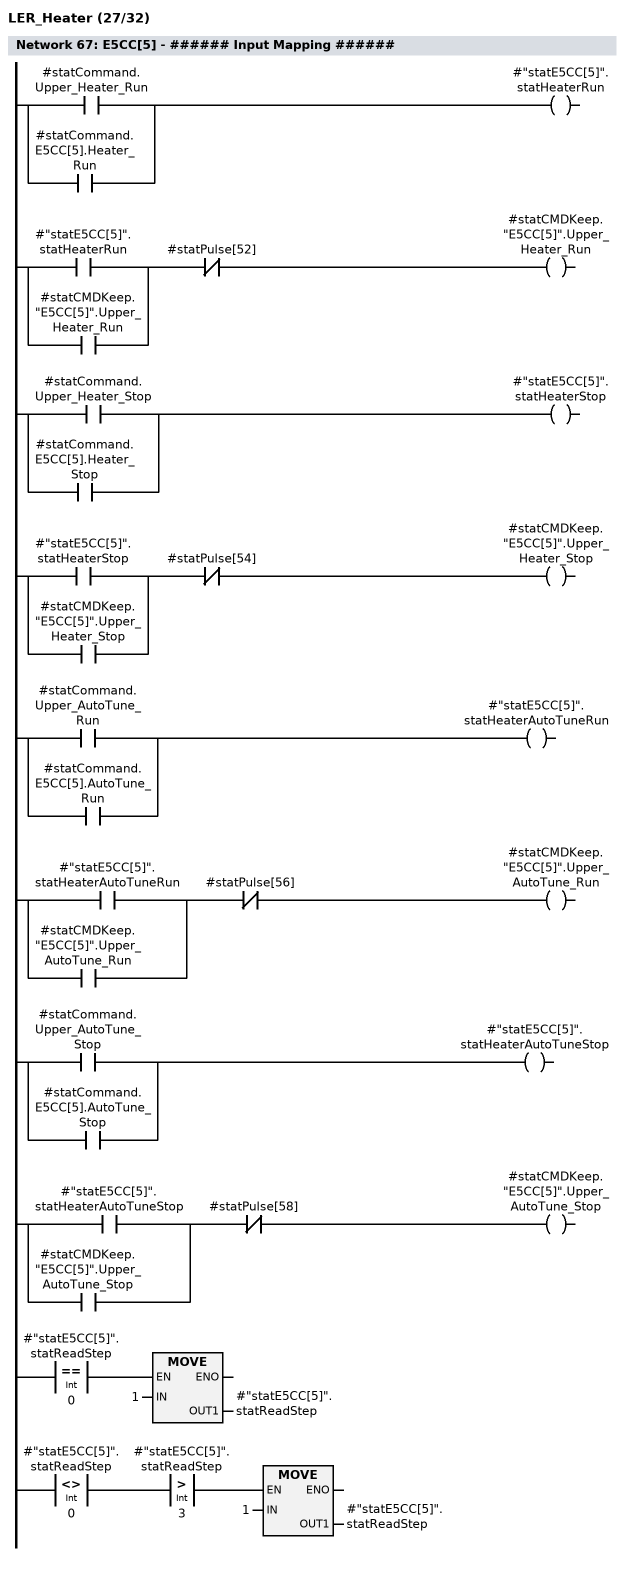
   RUNG wire#powerrail
      Contact( #statCommand.Upper_Heater_Run )
      wire#w1
      Coil( #"statE5CC[5]".statHeaterRun )
   END_RUNG
   RUNG wire#powerrail
      Contact( #statCommand.E5CC[5].Heater_Run )
   END_RUNG wire#w1
   RUNG wire#powerrail
      Contact( #"statE5CC[5]".statHeaterRun )
      wire#w2
      I_Contact( #statPulse[52] )
      Coil( #statCMDKeep."E5CC[5]".Upper_Heater_Run )
   END_RUNG
   RUNG wire#powerrail
      Contact( #statCMDKeep."E5CC[5]".Upper_Heater_Run )
   END_RUNG wire#w2
   RUNG wire#powerrail
      Contact( #statCommand.Upper_Heater_Stop )
      wire#w3
      Coil( #"statE5CC[5]".statHeaterStop )
   END_RUNG
   RUNG wire#powerrail
      Contact( #statCommand.E5CC[5].Heater_Stop )
   END_RUNG wire#w3
   RUNG wire#powerrail
      Contact( #"statE5CC[5]".statHeaterStop )
      wire#w4
      I_Contact( #statPulse[54] )
      Coil( #statCMDKeep."E5CC[5]".Upper_Heater_Stop )
   END_RUNG
   RUNG wire#powerrail
      Contact( #statCMDKeep."E5CC[5]".Upper_Heater_Stop )
   END_RUNG wire#w4
   RUNG wire#powerrail
      Contact( #statCommand.Upper_AutoTune_Run )
      wire#w5
      Coil( #"statE5CC[5]".statHeaterAutoTuneRun )
   END_RUNG
   RUNG wire#powerrail
      Contact( #statCommand.E5CC[5].AutoTune_Run )
   END_RUNG wire#w5
   RUNG wire#powerrail
      Contact( #"statE5CC[5]".statHeaterAutoTuneRun )
      wire#w6
      I_Contact( #statPulse[56] )
      Coil( #statCMDKeep."E5CC[5]".Upper_AutoTune_Run )
   END_RUNG
   RUNG wire#powerrail
      Contact( #statCMDKeep."E5CC[5]".Upper_AutoTune_Run )
   END_RUNG wire#w6
   RUNG wire#powerrail
      Contact( #statCommand.Upper_AutoTune_Stop )
      wire#w7
      Coil( #"statE5CC[5]".statHeaterAutoTuneStop )
   END_RUNG
   RUNG wire#powerrail
      Contact( #statCommand.E5CC[5].AutoTune_Stop )
   END_RUNG wire#w7
   RUNG wire#powerrail
      Contact( #"statE5CC[5]".statHeaterAutoTuneStop )
      wire#w8
      I_Contact( #statPulse[58] )
      Coil( #statCMDKeep."E5CC[5]".Upper_AutoTune_Stop )
   END_RUNG
   RUNG wire#powerrail
      Contact( #statCMDKeep."E5CC[5]".Upper_AutoTune_Stop )
   END_RUNG wire#w8
   RUNG wire#powerrail
      { S7_Templates := "SrcType := Int" } EQ_Contact(in1 := #"statE5CC[5]".statReadStep, in2 := 0)
      Move(in := 1, out1 => #"statE5CC[5]".statReadStep)
   END_RUNG
   RUNG wire#powerrail
      { S7_Templates := "SrcType := Int" } NE_Contact(in1 := #"statE5CC[5]".statReadStep, in2 := 0)
      { S7_Templates := "SrcType := Int" } GT_Contact(in1 := #"statE5CC[5]".statReadStep, in2 := 3)
      Move(in := 1, out1 => #"statE5CC[5]".statReadStep)
   END_RUNG
   // the same network as SCL:
   #"statE5CC[5]".statHeaterRun := #statCommand.Upper_Heater_Run OR #statCommand.E5CC[5].Heater_Run;
   #statCMDKeep."E5CC[5]".Upper_Heater_Run := (#"statE5CC[5]".statHeaterRun OR #statCMDKeep."E5CC[5]".Upper_Heater_Run) AND NOT #statPulse[52];
   #"statE5CC[5]".statHeaterStop := #statCommand.Upper_Heater_Stop OR #statCommand.E5CC[5].Heater_Stop;
   #statCMDKeep."E5CC[5]".Upper_Heater_Stop := (#"statE5CC[5]".statHeaterStop OR #statCMDKeep."E5CC[5]".Upper_Heater_Stop) AND NOT #statPulse[54];
   #"statE5CC[5]".statHeaterAutoTuneRun := #statCommand.Upper_AutoTune_Run OR #statCommand.E5CC[5].AutoTune_Run;
   #statCMDKeep."E5CC[5]".Upper_AutoTune_Run := (#"statE5CC[5]".statHeaterAutoTuneRun OR #statCMDKeep."E5CC[5]".Upper_AutoTune_Run) AND NOT #statPulse[56];
   #"statE5CC[5]".statHeaterAutoTuneStop := #statCommand.Upper_AutoTune_Stop OR #statCommand.E5CC[5].AutoTune_Stop;
   #statCMDKeep."E5CC[5]".Upper_AutoTune_Stop := (#"statE5CC[5]".statHeaterAutoTuneStop OR #statCMDKeep."E5CC[5]".Upper_AutoTune_Stop) AND NOT #statPulse[58];
   IF #"statE5CC[5]".statReadStep = 0 THEN #"statE5CC[5]".statReadStep := 1; END_IF;
   IF (#"statE5CC[5]".statReadStep <> 0) AND (#"statE5CC[5]".statReadStep > 3) THEN
       #"statE5CC[5]".statReadStep := 1;
   END_IF;
END_REGION

REGION Network 68: E5CC[5] -Read Temp PV + Status Command
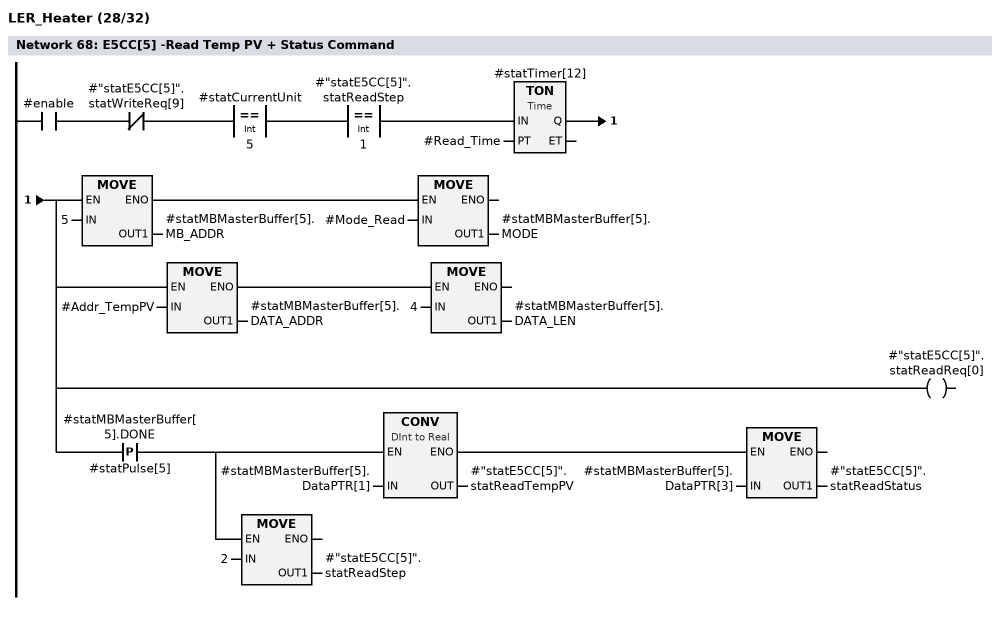
   RUNG wire#powerrail
      Contact( #enable )
      I_Contact( #"statE5CC[5]".statWriteReq[9] )
      { S7_Templates := "SrcType := Int" } EQ_Contact(in1 := #statCurrentUnit, in2 := 5)
      { S7_Templates := "SrcType := Int" } EQ_Contact(in1 := #"statE5CC[5]".statReadStep, in2 := 1)
      { S7_Templates := "time_type := Time" } #statTimer[12].TON(pt := #Read_Time, et =>)
      wire#w1
      Move(in := 5, out1 => #statMBMasterBuffer[5].MB_ADDR)
      Move(in := #Mode_Read, out1 => #statMBMasterBuffer[5].MODE)
   END_RUNG
   RUNG wire#w1
      Move(in := #Addr_TempPV, out1 => #statMBMasterBuffer[5].DATA_ADDR)
      Move(in := 4, out1 => #statMBMasterBuffer[5].DATA_LEN)
   END_RUNG
   RUNG wire#w1
      Coil( #"statE5CC[5]".statReadReq[0] )
   END_RUNG
   RUNG wire#w1
      P_Contact(operand := #statMBMasterBuffer[5].DONE, bit := #statPulse[5])
      wire#w2
      { S7_Templates := "[SrcType := DInt, DestType := Real]" } Convert(in := #statMBMasterBuffer[5].DataPTR[1], out => #"statE5CC[5]".statReadTempPV)
      Move(in := #statMBMasterBuffer[5].DataPTR[3], out1 => #"statE5CC[5]".statReadStatus)
   END_RUNG
   RUNG wire#w2
      Move(in := 2, out1 => #"statE5CC[5]".statReadStep)
   END_RUNG
   // the same network as SCL:
   #statTimer[12].TON(IN := #enable AND NOT #"statE5CC[5]".statWriteReq[9] AND (#statCurrentUnit = 5) AND (#"statE5CC[5]".statReadStep = 1),
                      PT := #Read_Time);
   IF #statTimer[12].Q THEN
       #statMBMasterBuffer[5].MB_ADDR := 5;
       #statMBMasterBuffer[5].MODE := #Mode_Read;
       #statMBMasterBuffer[5].DATA_ADDR := #Addr_TempPV;
       #statMBMasterBuffer[5].DATA_LEN := 4;
   END_IF;
   #"statE5CC[5]".statReadReq[0] := #statTimer[12].Q;
   #_w1 := #statTimer[12].Q AND #statMBMasterBuffer[5].DONE AND NOT #statPulse[5];   // rising edge of #statMBMasterBuffer[5].DONE
   #statPulse[5] := #statMBMasterBuffer[5].DONE;
   IF #_w1 THEN
       #"statE5CC[5]".statReadTempPV := DINT_TO_REAL(#statMBMasterBuffer[5].DataPTR[1]);
       #"statE5CC[5]".statReadStatus := #statMBMasterBuffer[5].DataPTR[3];
       #"statE5CC[5]".statReadStep := 2;
   END_IF;
END_REGION

REGION Network 69: E5CC[5] -Read TempSP + AlarmValue1 ~ AlarmValue2_LowerLimit Commad
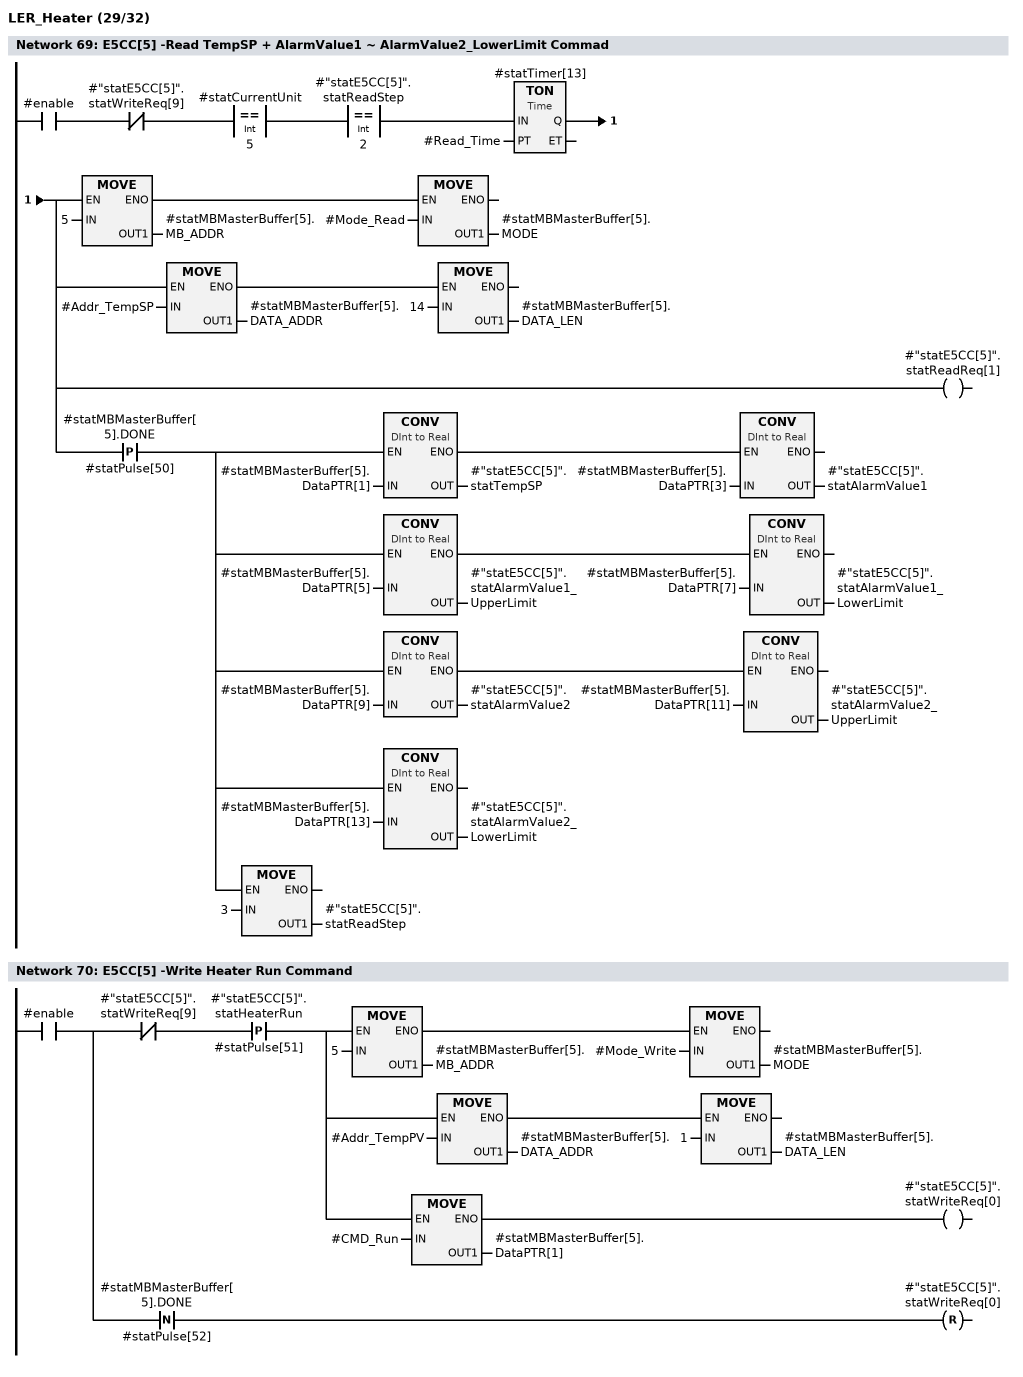
   RUNG wire#powerrail
      Contact( #enable )
      I_Contact( #"statE5CC[5]".statWriteReq[9] )
      { S7_Templates := "SrcType := Int" } EQ_Contact(in1 := #statCurrentUnit, in2 := 5)
      { S7_Templates := "SrcType := Int" } EQ_Contact(in1 := #"statE5CC[5]".statReadStep, in2 := 2)
      { S7_Templates := "time_type := Time" } #statTimer[13].TON(pt := #Read_Time, et =>)
      wire#w1
      Move(in := 5, out1 => #statMBMasterBuffer[5].MB_ADDR)
      Move(in := #Mode_Read, out1 => #statMBMasterBuffer[5].MODE)
   END_RUNG
   RUNG wire#w1
      Move(in := #Addr_TempSP, out1 => #statMBMasterBuffer[5].DATA_ADDR)
      Move(in := 14, out1 => #statMBMasterBuffer[5].DATA_LEN)
   END_RUNG
   RUNG wire#w1
      Coil( #"statE5CC[5]".statReadReq[1] )
   END_RUNG
   RUNG wire#w1
      P_Contact(operand := #statMBMasterBuffer[5].DONE, bit := #statPulse[50])
      wire#w2
      { S7_Templates := "[SrcType := DInt, DestType := Real]" } Convert(in := #statMBMasterBuffer[5].DataPTR[1], out => #"statE5CC[5]".statTempSP)
      { S7_Templates := "[SrcType := DInt, DestType := Real]" } Convert(in := #statMBMasterBuffer[5].DataPTR[3], out => #"statE5CC[5]".statAlarmValue1)
   END_RUNG
   RUNG wire#w2
      { S7_Templates := "[SrcType := DInt, DestType := Real]" } Convert(in := #statMBMasterBuffer[5].DataPTR[5], out => #"statE5CC[5]".statAlarmValue1_UpperLimit)
      { S7_Templates := "[SrcType := DInt, DestType := Real]" } Convert(in := #statMBMasterBuffer[5].DataPTR[7], out => #"statE5CC[5]".statAlarmValue1_LowerLimit)
   END_RUNG
   RUNG wire#w2
      { S7_Templates := "[SrcType := DInt, DestType := Real]" } Convert(in := #statMBMasterBuffer[5].DataPTR[9], out => #"statE5CC[5]".statAlarmValue2)
      { S7_Templates := "[SrcType := DInt, DestType := Real]" } Convert(in := #statMBMasterBuffer[5].DataPTR[11], out => #"statE5CC[5]".statAlarmValue2_UpperLimit)
   END_RUNG
   RUNG wire#w2
      { S7_Templates := "[SrcType := DInt, DestType := Real]" } Convert(in := #statMBMasterBuffer[5].DataPTR[13], out => #"statE5CC[5]".statAlarmValue2_LowerLimit)
   END_RUNG
   RUNG wire#w2
      Move(in := 3, out1 => #"statE5CC[5]".statReadStep)
   END_RUNG
   // the same network as SCL:
   #statTimer[13].TON(IN := #enable AND NOT #"statE5CC[5]".statWriteReq[9] AND (#statCurrentUnit = 5) AND (#"statE5CC[5]".statReadStep = 2),
                      PT := #Read_Time);
   IF #statTimer[13].Q THEN
       #statMBMasterBuffer[5].MB_ADDR := 5;
       #statMBMasterBuffer[5].MODE := #Mode_Read;
       #statMBMasterBuffer[5].DATA_ADDR := #Addr_TempSP;
       #statMBMasterBuffer[5].DATA_LEN := 14;
   END_IF;
   #"statE5CC[5]".statReadReq[1] := #statTimer[13].Q;
   #_w1 := #statTimer[13].Q AND #statMBMasterBuffer[5].DONE AND NOT #statPulse[50];   // rising edge of #statMBMasterBuffer[5].DONE
   #statPulse[50] := #statMBMasterBuffer[5].DONE;
   IF #_w1 THEN
       #"statE5CC[5]".statTempSP := DINT_TO_REAL(#statMBMasterBuffer[5].DataPTR[1]);
       #"statE5CC[5]".statAlarmValue1 := DINT_TO_REAL(#statMBMasterBuffer[5].DataPTR[3]);
       #"statE5CC[5]".statAlarmValue1_UpperLimit := DINT_TO_REAL(#statMBMasterBuffer[5].DataPTR[5]);
       #"statE5CC[5]".statAlarmValue1_LowerLimit := DINT_TO_REAL(#statMBMasterBuffer[5].DataPTR[7]);
       #"statE5CC[5]".statAlarmValue2 := DINT_TO_REAL(#statMBMasterBuffer[5].DataPTR[9]);
       #"statE5CC[5]".statAlarmValue2_UpperLimit := DINT_TO_REAL(#statMBMasterBuffer[5].DataPTR[11]);
       #"statE5CC[5]".statAlarmValue2_LowerLimit := DINT_TO_REAL(#statMBMasterBuffer[5].DataPTR[13]);
       #"statE5CC[5]".statReadStep := 3;
   END_IF;
END_REGION

REGION Network 70: E5CC[5] -Write Heater Run Command
   RUNG wire#powerrail
      Contact( #enable )
      wire#w1
      I_Contact( #"statE5CC[5]".statWriteReq[9] )
      P_Contact(operand := #"statE5CC[5]".statHeaterRun, bit := #statPulse[51])
      wire#w2
      Move(in := 5, out1 => #statMBMasterBuffer[5].MB_ADDR)
      Move(in := #Mode_Write, out1 => #statMBMasterBuffer[5].MODE)
   END_RUNG
   RUNG wire#w2
      Move(in := #Addr_TempPV, out1 => #statMBMasterBuffer[5].DATA_ADDR)
      Move(in := 1, out1 => #statMBMasterBuffer[5].DATA_LEN)
   END_RUNG
   RUNG wire#w2
      Move(in := #CMD_Run, out1 => #statMBMasterBuffer[5].DataPTR[1])
      Coil( #"statE5CC[5]".statWriteReq[0] )
   END_RUNG
   RUNG wire#w1
      N_Contact(operand := #statMBMasterBuffer[5].DONE, bit := #statPulse[52])
      R_Coil( #"statE5CC[5]".statWriteReq[0] )
   END_RUNG
   // the same network as SCL:
   #_w1 := #enable AND NOT #"statE5CC[5]".statWriteReq[9] AND #"statE5CC[5]".statHeaterRun AND NOT #statPulse[51];   // rising edge of #"statE5CC[5]".statHeaterRun
   #statPulse[51] := #"statE5CC[5]".statHeaterRun;
   IF #_w1 THEN
       #statMBMasterBuffer[5].MB_ADDR := 5;
       #statMBMasterBuffer[5].MODE := #Mode_Write;
       #statMBMasterBuffer[5].DATA_ADDR := #Addr_TempPV;
       #statMBMasterBuffer[5].DATA_LEN := 1;
       #statMBMasterBuffer[5].DataPTR[1] := #CMD_Run;
   END_IF;
   #"statE5CC[5]".statWriteReq[0] := #_w1;
   #_w2 := #enable AND NOT #statMBMasterBuffer[5].DONE AND #statPulse[52];   // falling edge of #statMBMasterBuffer[5].DONE
   #statPulse[52] := #statMBMasterBuffer[5].DONE;
   IF #_w2 THEN #"statE5CC[5]".statWriteReq[0] := FALSE; END_IF;
END_REGION

REGION Network 71: E5CC[5] -Write Heater Stop Command
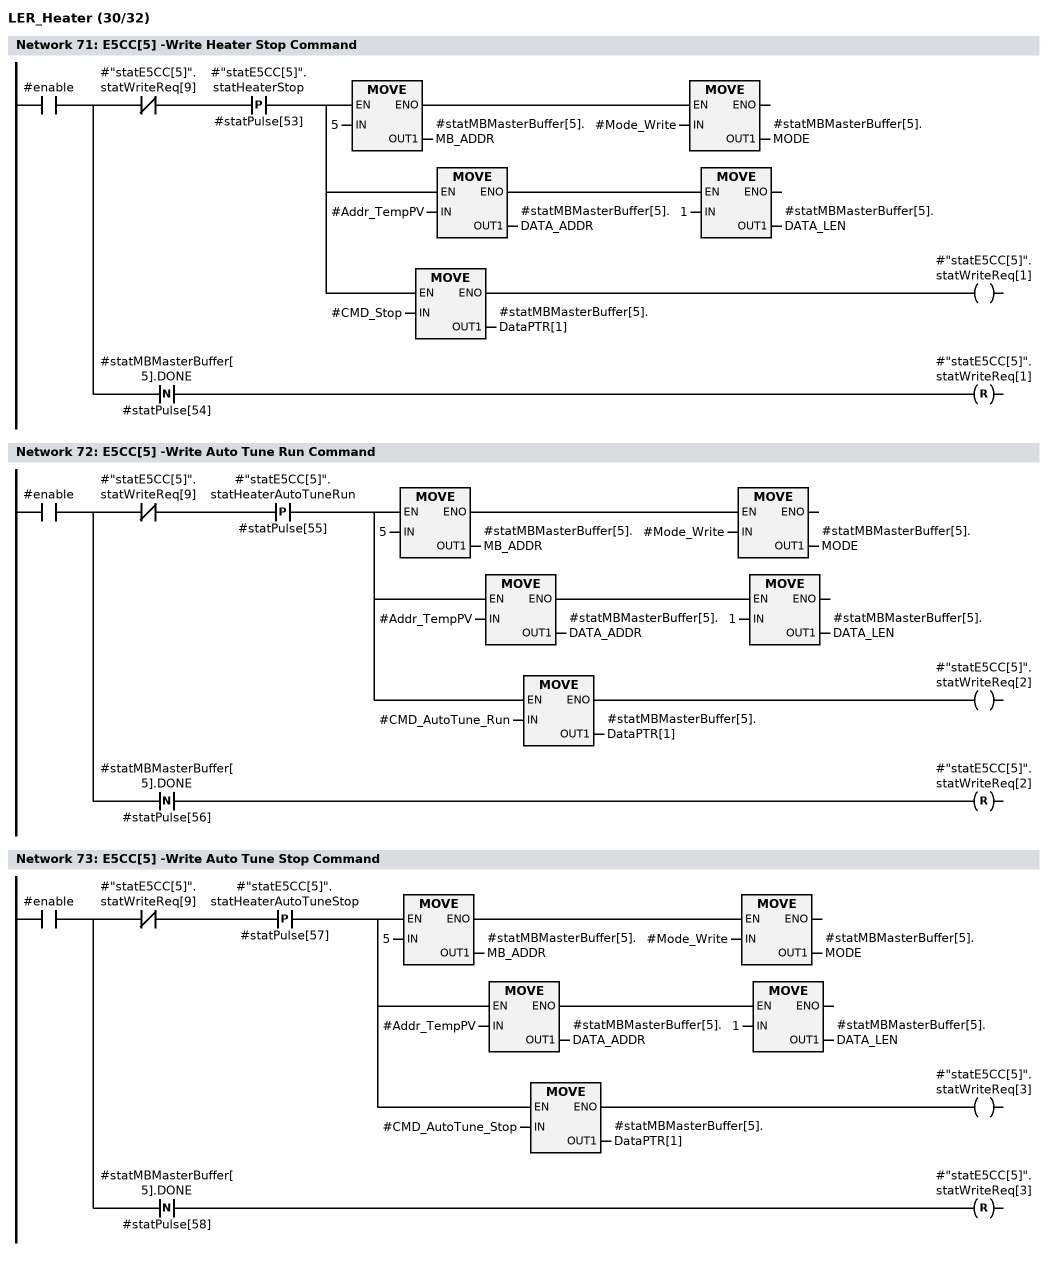
   RUNG wire#powerrail
      Contact( #enable )
      wire#w1
      I_Contact( #"statE5CC[5]".statWriteReq[9] )
      P_Contact(operand := #"statE5CC[5]".statHeaterStop, bit := #statPulse[53])
      wire#w2
      Move(in := 5, out1 => #statMBMasterBuffer[5].MB_ADDR)
      Move(in := #Mode_Write, out1 => #statMBMasterBuffer[5].MODE)
   END_RUNG
   RUNG wire#w2
      Move(in := #Addr_TempPV, out1 => #statMBMasterBuffer[5].DATA_ADDR)
      Move(in := 1, out1 => #statMBMasterBuffer[5].DATA_LEN)
   END_RUNG
   RUNG wire#w2
      Move(in := #CMD_Stop, out1 => #statMBMasterBuffer[5].DataPTR[1])
      Coil( #"statE5CC[5]".statWriteReq[1] )
   END_RUNG
   RUNG wire#w1
      N_Contact(operand := #statMBMasterBuffer[5].DONE, bit := #statPulse[54])
      R_Coil( #"statE5CC[5]".statWriteReq[1] )
   END_RUNG
   // the same network as SCL:
   #_w1 := #enable AND NOT #"statE5CC[5]".statWriteReq[9] AND #"statE5CC[5]".statHeaterStop AND NOT #statPulse[53];   // rising edge of #"statE5CC[5]".statHeaterStop
   #statPulse[53] := #"statE5CC[5]".statHeaterStop;
   IF #_w1 THEN
       #statMBMasterBuffer[5].MB_ADDR := 5;
       #statMBMasterBuffer[5].MODE := #Mode_Write;
       #statMBMasterBuffer[5].DATA_ADDR := #Addr_TempPV;
       #statMBMasterBuffer[5].DATA_LEN := 1;
       #statMBMasterBuffer[5].DataPTR[1] := #CMD_Stop;
   END_IF;
   #"statE5CC[5]".statWriteReq[1] := #_w1;
   #_w2 := #enable AND NOT #statMBMasterBuffer[5].DONE AND #statPulse[54];   // falling edge of #statMBMasterBuffer[5].DONE
   #statPulse[54] := #statMBMasterBuffer[5].DONE;
   IF #_w2 THEN #"statE5CC[5]".statWriteReq[1] := FALSE; END_IF;
END_REGION

REGION Network 72: E5CC[5] -Write Auto Tune Run Command
   RUNG wire#powerrail
      Contact( #enable )
      wire#w1
      I_Contact( #"statE5CC[5]".statWriteReq[9] )
      P_Contact(operand := #"statE5CC[5]".statHeaterAutoTuneRun, bit := #statPulse[55])
      wire#w2
      Move(in := 5, out1 => #statMBMasterBuffer[5].MB_ADDR)
      Move(in := #Mode_Write, out1 => #statMBMasterBuffer[5].MODE)
   END_RUNG
   RUNG wire#w2
      Move(in := #Addr_TempPV, out1 => #statMBMasterBuffer[5].DATA_ADDR)
      Move(in := 1, out1 => #statMBMasterBuffer[5].DATA_LEN)
   END_RUNG
   RUNG wire#w2
      Move(in := #CMD_AutoTune_Run, out1 => #statMBMasterBuffer[5].DataPTR[1])
      Coil( #"statE5CC[5]".statWriteReq[2] )
   END_RUNG
   RUNG wire#w1
      N_Contact(operand := #statMBMasterBuffer[5].DONE, bit := #statPulse[56])
      R_Coil( #"statE5CC[5]".statWriteReq[2] )
   END_RUNG
   // the same network as SCL:
   #_w1 := #enable AND NOT #"statE5CC[5]".statWriteReq[9] AND #"statE5CC[5]".statHeaterAutoTuneRun AND NOT #statPulse[55];   // rising edge of #"statE5CC[5]".statHeaterAutoTuneRun
   #statPulse[55] := #"statE5CC[5]".statHeaterAutoTuneRun;
   IF #_w1 THEN
       #statMBMasterBuffer[5].MB_ADDR := 5;
       #statMBMasterBuffer[5].MODE := #Mode_Write;
       #statMBMasterBuffer[5].DATA_ADDR := #Addr_TempPV;
       #statMBMasterBuffer[5].DATA_LEN := 1;
       #statMBMasterBuffer[5].DataPTR[1] := #CMD_AutoTune_Run;
   END_IF;
   #"statE5CC[5]".statWriteReq[2] := #_w1;
   #_w2 := #enable AND NOT #statMBMasterBuffer[5].DONE AND #statPulse[56];   // falling edge of #statMBMasterBuffer[5].DONE
   #statPulse[56] := #statMBMasterBuffer[5].DONE;
   IF #_w2 THEN #"statE5CC[5]".statWriteReq[2] := FALSE; END_IF;
END_REGION

REGION Network 73: E5CC[5] -Write Auto Tune Stop Command
   RUNG wire#powerrail
      Contact( #enable )
      wire#w1
      I_Contact( #"statE5CC[5]".statWriteReq[9] )
      P_Contact(operand := #"statE5CC[5]".statHeaterAutoTuneStop, bit := #statPulse[57])
      wire#w2
      Move(in := 5, out1 => #statMBMasterBuffer[5].MB_ADDR)
      Move(in := #Mode_Write, out1 => #statMBMasterBuffer[5].MODE)
   END_RUNG
   RUNG wire#w2
      Move(in := #Addr_TempPV, out1 => #statMBMasterBuffer[5].DATA_ADDR)
      Move(in := 1, out1 => #statMBMasterBuffer[5].DATA_LEN)
   END_RUNG
   RUNG wire#w2
      Move(in := #CMD_AutoTune_Stop, out1 => #statMBMasterBuffer[5].DataPTR[1])
      Coil( #"statE5CC[5]".statWriteReq[3] )
   END_RUNG
   RUNG wire#w1
      N_Contact(operand := #statMBMasterBuffer[5].DONE, bit := #statPulse[58])
      R_Coil( #"statE5CC[5]".statWriteReq[3] )
   END_RUNG
   // the same network as SCL:
   #_w1 := #enable AND NOT #"statE5CC[5]".statWriteReq[9] AND #"statE5CC[5]".statHeaterAutoTuneStop AND NOT #statPulse[57];   // rising edge of #"statE5CC[5]".statHeaterAutoTuneStop
   #statPulse[57] := #"statE5CC[5]".statHeaterAutoTuneStop;
   IF #_w1 THEN
       #statMBMasterBuffer[5].MB_ADDR := 5;
       #statMBMasterBuffer[5].MODE := #Mode_Write;
       #statMBMasterBuffer[5].DATA_ADDR := #Addr_TempPV;
       #statMBMasterBuffer[5].DATA_LEN := 1;
       #statMBMasterBuffer[5].DataPTR[1] := #CMD_AutoTune_Stop;
   END_IF;
   #"statE5CC[5]".statWriteReq[3] := #_w1;
   #_w2 := #enable AND NOT #statMBMasterBuffer[5].DONE AND #statPulse[58];   // falling edge of #statMBMasterBuffer[5].DONE
   #statPulse[58] := #statMBMasterBuffer[5].DONE;
   IF #_w2 THEN #"statE5CC[5]".statWriteReq[3] := FALSE; END_IF;
END_REGION

REGION Network 74: E5CC[5]-Write TempSP + AlarmValue1 ~ AlarmValue2_LowerLimit Command
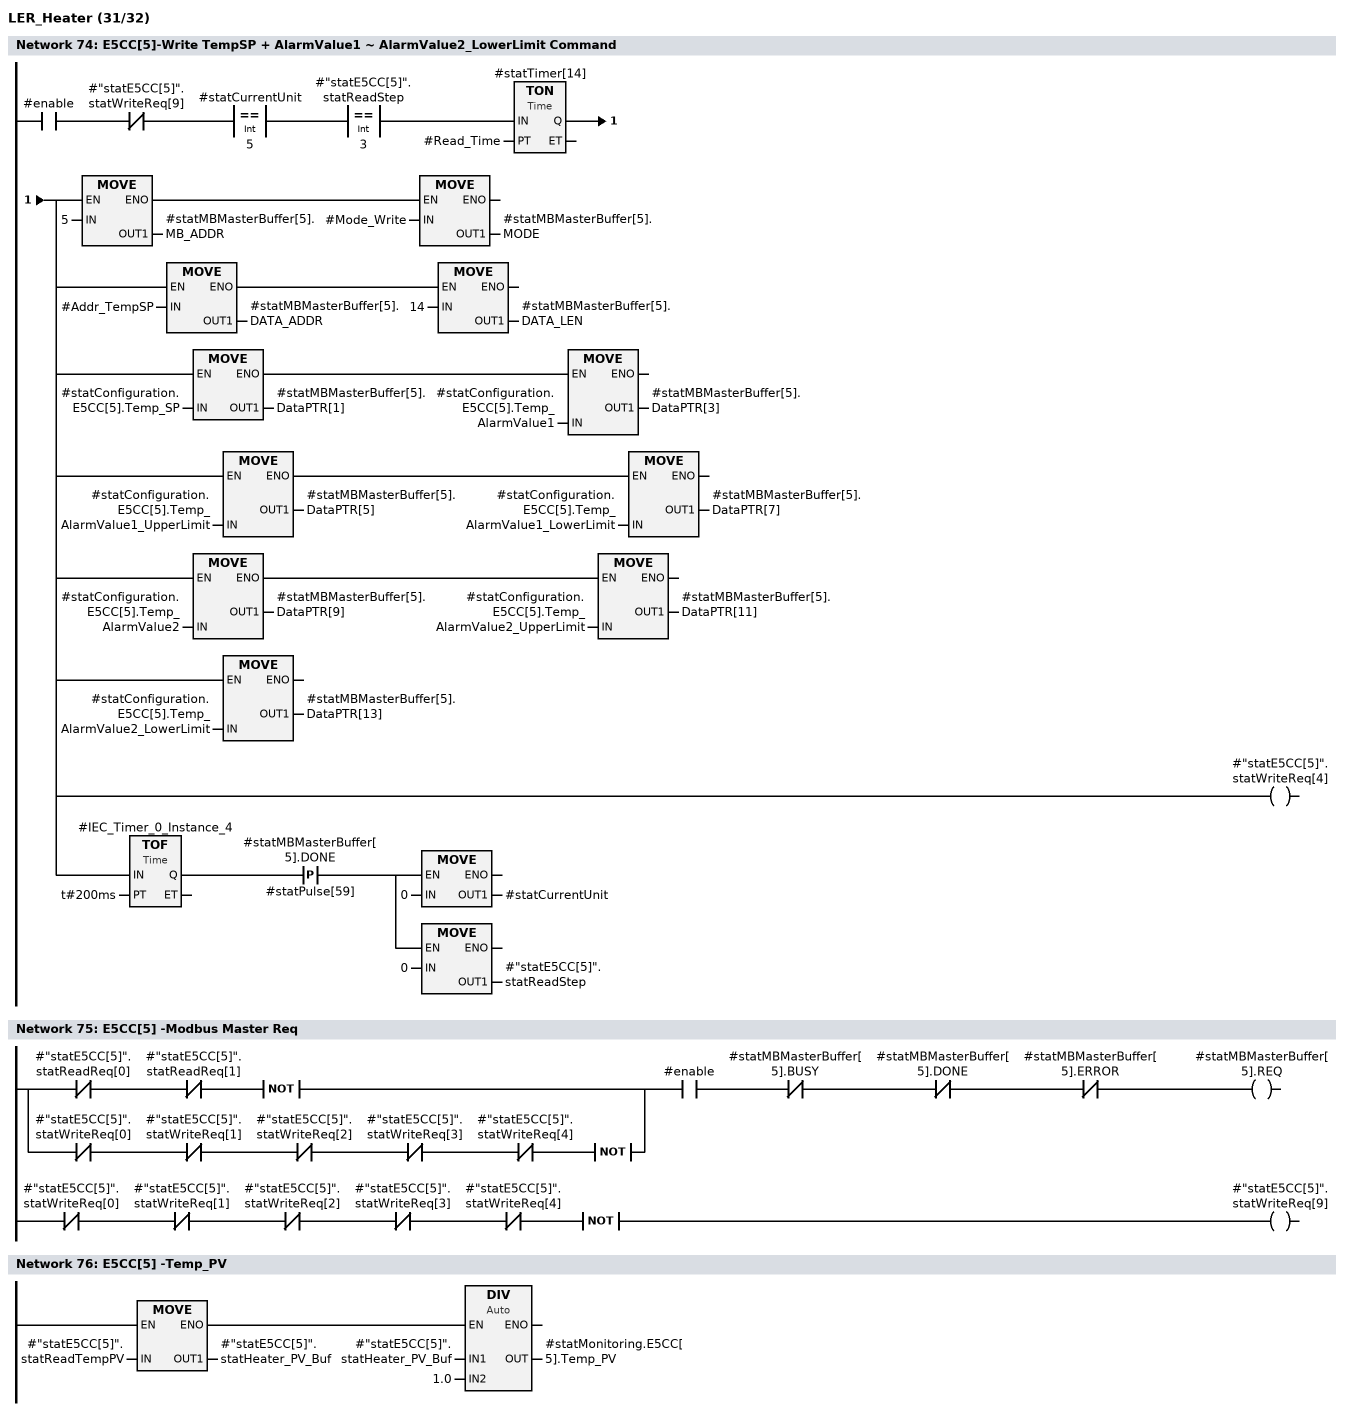
   RUNG wire#powerrail
      Contact( #enable )
      I_Contact( #"statE5CC[5]".statWriteReq[9] )
      { S7_Templates := "SrcType := Int" } EQ_Contact(in1 := #statCurrentUnit, in2 := 5)
      { S7_Templates := "SrcType := Int" } EQ_Contact(in1 := #"statE5CC[5]".statReadStep, in2 := 3)
      { S7_Templates := "time_type := Time" } #statTimer[14].TON(pt := #Read_Time, et =>)
      wire#w1
      Move(in := 5, out1 => #statMBMasterBuffer[5].MB_ADDR)
      Move(in := #Mode_Write, out1 => #statMBMasterBuffer[5].MODE)
   END_RUNG
   RUNG wire#w1
      Move(in := #Addr_TempSP, out1 => #statMBMasterBuffer[5].DATA_ADDR)
      Move(in := 14, out1 => #statMBMasterBuffer[5].DATA_LEN)
   END_RUNG
   RUNG wire#w1
      Move(in := #statConfiguration.E5CC[5].Temp_SP, out1 => #statMBMasterBuffer[5].DataPTR[1])
      Move(in := #statConfiguration.E5CC[5].Temp_AlarmValue1, out1 => #statMBMasterBuffer[5].DataPTR[3])
   END_RUNG
   RUNG wire#w1
      Move(in := #statConfiguration.E5CC[5].Temp_AlarmValue1_UpperLimit, out1 => #statMBMasterBuffer[5].DataPTR[5])
      Move(in := #statConfiguration.E5CC[5].Temp_AlarmValue1_LowerLimit, out1 => #statMBMasterBuffer[5].DataPTR[7])
   END_RUNG
   RUNG wire#w1
      Move(in := #statConfiguration.E5CC[5].Temp_AlarmValue2, out1 => #statMBMasterBuffer[5].DataPTR[9])
      Move(in := #statConfiguration.E5CC[5].Temp_AlarmValue2_UpperLimit, out1 => #statMBMasterBuffer[5].DataPTR[11])
   END_RUNG
   RUNG wire#w1
      Move(in := #statConfiguration.E5CC[5].Temp_AlarmValue2_LowerLimit, out1 => #statMBMasterBuffer[5].DataPTR[13])
   END_RUNG
   RUNG wire#w1
      Coil( #"statE5CC[5]".statWriteReq[4] )
   END_RUNG
   RUNG wire#w1
      { S7_Templates := "time_type := Time" } #IEC_Timer_0_Instance_4.TOF(pt := t#200ms, et =>)
      P_Contact(operand := #statMBMasterBuffer[5].DONE, bit := #statPulse[59])
      wire#w2
      Move(in := 0, out1 => #statCurrentUnit)
   END_RUNG
   RUNG wire#w2
      Move(in := 0, out1 => #"statE5CC[5]".statReadStep)
   END_RUNG
   // the same network as SCL:
   #statTimer[14].TON(IN := #enable AND NOT #"statE5CC[5]".statWriteReq[9] AND (#statCurrentUnit = 5) AND (#"statE5CC[5]".statReadStep = 3),
                      PT := #Read_Time);
   IF #statTimer[14].Q THEN
       #statMBMasterBuffer[5].MB_ADDR := 5;
       #statMBMasterBuffer[5].MODE := #Mode_Write;
       #statMBMasterBuffer[5].DATA_ADDR := #Addr_TempSP;
       #statMBMasterBuffer[5].DATA_LEN := 14;
       #statMBMasterBuffer[5].DataPTR[1] := #statConfiguration.E5CC[5].Temp_SP;
       #statMBMasterBuffer[5].DataPTR[3] := #statConfiguration.E5CC[5].Temp_AlarmValue1;
       #statMBMasterBuffer[5].DataPTR[5] := #statConfiguration.E5CC[5].Temp_AlarmValue1_UpperLimit;
       #statMBMasterBuffer[5].DataPTR[7] := #statConfiguration.E5CC[5].Temp_AlarmValue1_LowerLimit;
       #statMBMasterBuffer[5].DataPTR[9] := #statConfiguration.E5CC[5].Temp_AlarmValue2;
       #statMBMasterBuffer[5].DataPTR[11] := #statConfiguration.E5CC[5].Temp_AlarmValue2_UpperLimit;
       #statMBMasterBuffer[5].DataPTR[13] := #statConfiguration.E5CC[5].Temp_AlarmValue2_LowerLimit;
   END_IF;
   #"statE5CC[5]".statWriteReq[4] := #statTimer[14].Q;
   #IEC_Timer_0_Instance_4(IN := #statTimer[14].Q, PT := t#200ms);   // TOF
   #_w1 := #IEC_Timer_0_Instance_4.Q AND #statMBMasterBuffer[5].DONE AND NOT #statPulse[59];   // rising edge of #statMBMasterBuffer[5].DONE
   #statPulse[59] := #statMBMasterBuffer[5].DONE;
   IF #_w1 THEN
       #statCurrentUnit := 0;
       #"statE5CC[5]".statReadStep := 0;
   END_IF;
END_REGION

REGION Network 75: E5CC[5] -Modbus Master Req
   RUNG wire#powerrail
      I_Contact( #"statE5CC[5]".statReadReq[0] )
      I_Contact( #"statE5CC[5]".statReadReq[1] )
      Not()
      wire#w1
      Contact( #enable )
      I_Contact( #statMBMasterBuffer[5].BUSY )
      I_Contact( #statMBMasterBuffer[5].DONE )
      I_Contact( #statMBMasterBuffer[5].ERROR )
      Coil( #statMBMasterBuffer[5].REQ )
   END_RUNG
   RUNG wire#powerrail
      I_Contact( #"statE5CC[5]".statWriteReq[0] )
      I_Contact( #"statE5CC[5]".statWriteReq[1] )
      I_Contact( #"statE5CC[5]".statWriteReq[2] )
      I_Contact( #"statE5CC[5]".statWriteReq[3] )
      I_Contact( #"statE5CC[5]".statWriteReq[4] )
      Not()
   END_RUNG wire#w1
   RUNG wire#powerrail
      I_Contact( #"statE5CC[5]".statWriteReq[0] )
      I_Contact( #"statE5CC[5]".statWriteReq[1] )
      I_Contact( #"statE5CC[5]".statWriteReq[2] )
      I_Contact( #"statE5CC[5]".statWriteReq[3] )
      I_Contact( #"statE5CC[5]".statWriteReq[4] )
      Not()
      Coil( #"statE5CC[5]".statWriteReq[9] )
   END_RUNG
   // the same network as SCL:
   #statMBMasterBuffer[5].REQ := (NOT (NOT #"statE5CC[5]".statReadReq[0] AND NOT #"statE5CC[5]".statReadReq[1]) OR NOT (NOT #"statE5CC[5]".statWriteReq[0] AND NOT #"statE5CC[5]".statWriteReq[1] AND NOT #"statE5CC[5]".statWriteReq[2] AND NOT #"statE5CC[5]".statWriteReq[3] AND NOT #"statE5CC[5]".statWriteReq[4])) AND #enable AND NOT #statMBMasterBuffer[5].BUSY AND NOT #statMBMasterBuffer[5].DONE AND NOT #statMBMasterBuffer[5].ERROR;
   #"statE5CC[5]".statWriteReq[9] := NOT (NOT #"statE5CC[5]".statWriteReq[0] AND NOT #"statE5CC[5]".statWriteReq[1] AND NOT #"statE5CC[5]".statWriteReq[2] AND NOT #"statE5CC[5]".statWriteReq[3] AND NOT #"statE5CC[5]".statWriteReq[4]);
END_REGION

REGION Network 76: E5CC[5] -Temp_PV
   RUNG wire#powerrail
      Move(in := #"statE5CC[5]".statReadTempPV, out1 => #"statE5CC[5]".statHeater_PV_Buf)
      Div(in1 := #"statE5CC[5]".statHeater_PV_Buf, in2 := 1.0, out => #statMonitoring.E5CC[5].Temp_PV)
   END_RUNG
   // the same network as SCL:
   #"statE5CC[5]".statHeater_PV_Buf := #"statE5CC[5]".statReadTempPV;
   #statMonitoring.E5CC[5].Temp_PV := #"statE5CC[5]".statHeater_PV_Buf / 1.0;
END_REGION

REGION Network 77: E5CC[5] -Temp_PV Complete Check
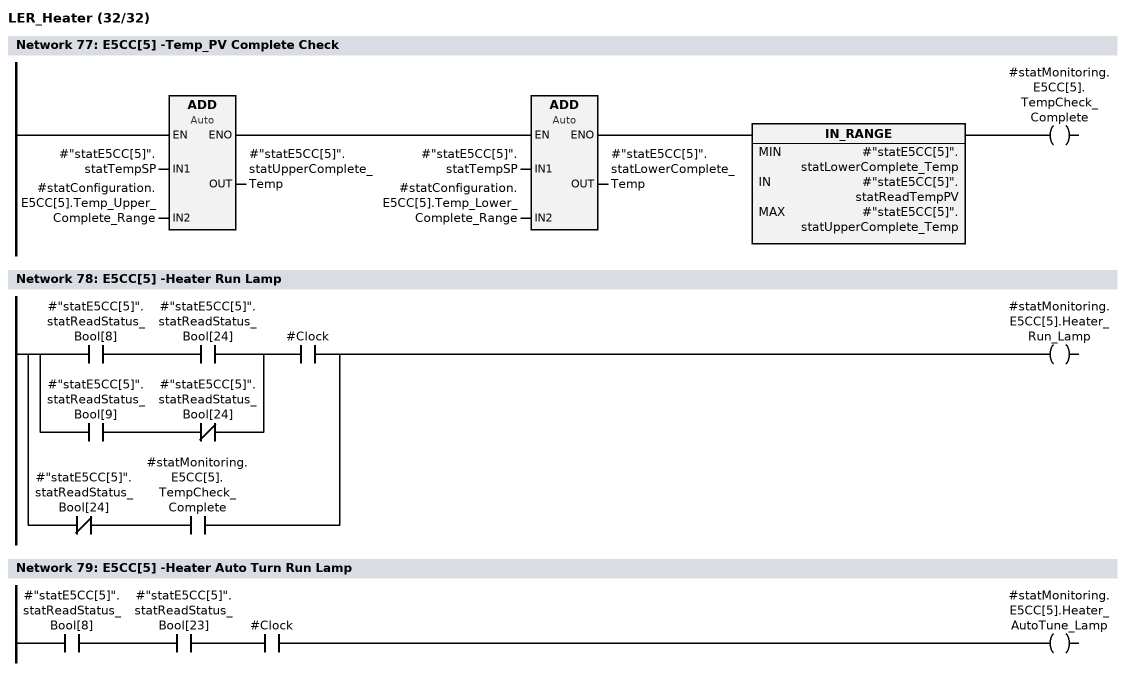
   RUNG wire#powerrail
      Add(in1 := #"statE5CC[5]".statTempSP, in2 := #statConfiguration.E5CC[5].Temp_Upper_Complete_Range, out => #"statE5CC[5]".statUpperComplete_Temp)
      Add(in1 := #"statE5CC[5]".statTempSP, in2 := #statConfiguration.E5CC[5].Temp_Lower_Complete_Range, out => #"statE5CC[5]".statLowerComplete_Temp)
      { S7_Templates := "SrcType := Real" } InRange(min := #"statE5CC[5]".statLowerComplete_Temp, in := #"statE5CC[5]".statReadTempPV, max := #"statE5CC[5]".statUpperComplete_Temp)
      Coil( #statMonitoring.E5CC[5].TempCheck_Complete )
   END_RUNG
   // the same network as SCL:
   #"statE5CC[5]".statUpperComplete_Temp := #"statE5CC[5]".statTempSP + #statConfiguration.E5CC[5].Temp_Upper_Complete_Range;
   #"statE5CC[5]".statLowerComplete_Temp := #"statE5CC[5]".statTempSP + #statConfiguration.E5CC[5].Temp_Lower_Complete_Range;
   #statMonitoring.E5CC[5].TempCheck_Complete := (#"statE5CC[5]".statLowerComplete_Temp <= #"statE5CC[5]".statReadTempPV) AND (#"statE5CC[5]".statReadTempPV <= #"statE5CC[5]".statUpperComplete_Temp);
END_REGION

REGION Network 78: E5CC[5] -Heater Run Lamp
   RUNG wire#powerrail
      Contact( #"statE5CC[5]".statReadStatus_Bool[8] )
      Contact( #"statE5CC[5]".statReadStatus_Bool[24] )
      wire#w1
      Contact( #Clock )
      wire#w2
      Coil( #statMonitoring.E5CC[5].Heater_Run_Lamp )
   END_RUNG
   RUNG wire#powerrail
      Contact( #"statE5CC[5]".statReadStatus_Bool[9] )
      I_Contact( #"statE5CC[5]".statReadStatus_Bool[24] )
   END_RUNG wire#w1
   RUNG wire#powerrail
      I_Contact( #"statE5CC[5]".statReadStatus_Bool[24] )
      Contact( #statMonitoring.E5CC[5].TempCheck_Complete )
   END_RUNG wire#w2
   // the same network as SCL:
   #statMonitoring.E5CC[5].Heater_Run_Lamp := (((#"statE5CC[5]".statReadStatus_Bool[8] AND #"statE5CC[5]".statReadStatus_Bool[24]) OR (#"statE5CC[5]".statReadStatus_Bool[9] AND NOT #"statE5CC[5]".statReadStatus_Bool[24])) AND #Clock) OR (NOT #"statE5CC[5]".statReadStatus_Bool[24] AND #statMonitoring.E5CC[5].TempCheck_Complete);
END_REGION

REGION Network 79: E5CC[5] -Heater Auto Turn Run Lamp
   RUNG wire#powerrail
      Contact( #"statE5CC[5]".statReadStatus_Bool[8] )
      Contact( #"statE5CC[5]".statReadStatus_Bool[23] )
      Contact( #Clock )
      Coil( #statMonitoring.E5CC[5].Heater_AutoTune_Lamp )
   END_RUNG
   // the same network as SCL:
   #statMonitoring.E5CC[5].Heater_AutoTune_Lamp := #"statE5CC[5]".statReadStatus_Bool[8] AND #"statE5CC[5]".statReadStatus_Bool[23] AND #Clock;
END_REGION

REGION Network 80 (SCL): E5CC[5] -Error Check
   REGION  E5CC Error Status
       // Dword to Bool
       SCATTER(IN := #"statE5CC[5]".statReadStatus,
               OUT => #"statE5CC[5]".statReadStatus_Bool);
   END_REGION


   REGION Error Code Search
       IF #"statE5CC[5]".statReadStatus <> 0 THEN
           CASE #"statE5CC[5]".statReadStatus OF
               #ERR_HEATER_CURRENT_VALUE_EXCEEDED_CT1:
                   #statMonitoring.E5CC[5].Status := #ERR_HEATER_CURRENT_VALUE_EXCEEDED_CT1;
               #ERR_HEATER_CURRENT_VALUE_HOLD_CT1:
                   #statMonitoring.E5CC[5].Status := #ERR_HEATER_CURRENT_VALUE_HOLD_CT1;
               #ERR_AD_CONVERTER_ABNORMALITY:
                   #statMonitoring.E5CC[5].Status := #ERR_AD_CONVERTER_ABNORMALITY;
               #ERR_HS_SSR_FAULT_ALERT_CT1:
                   #statMonitoring.E5CC[5].Status := #ERR_HS_SSR_FAULT_ALERT_CT1;
               #ERR_RSP_INPUT_ABNORMALITIES:
                   #statMonitoring.E5CC[5].Status := #ERR_RSP_INPUT_ABNORMALITIES;
               #ERR_MORE_THAN_INPUT:
                   #statMonitoring.E5CC[5].Status := #ERR_MORE_THAN_INPUT;
               #ERR_POTENTIOMETER_INPUT_ABNORMAL:
                   #statMonitoring.E5CC[5].Status := #ERR_POTENTIOMETER_INPUT_ABNORMAL;
               #ERR_CONTROL_OUTPUT_HEATED_OPEN_OUTPUT:
                   #statMonitoring.E5CC[5].Status := #ERR_CONTROL_OUTPUT_HEATED_OPEN_OUTPUT;
               #ERR_CONTROL_OUTPUT_COOL_CLOSE_OUTPUT:
                   #statMonitoring.E5CC[5].Status := #ERR_CONTROL_OUTPUT_COOL_CLOSE_OUTPUT;
               #ERR_HEATER_OPEN_CIRCUIT_HB_ALARM_CT1:
                   #statMonitoring.E5CC[5].Status := #ERR_HEATER_OPEN_CIRCUIT_HB_ALARM_CT1;
               #ERR_HEATER_OPEN_CIRCUIT_HB_ALARM_CT2:
                   #statMonitoring.E5CC[5].Status := #ERR_HEATER_OPEN_CIRCUIT_HB_ALARM_CT2;
               #ERR_ALERT_1:
                   #statMonitoring.E5CC[5].Status := #ERR_ALERT_1;
               #ERR_ALERT_2:
                   #statMonitoring.E5CC[5].Status := #ERR_ALERT_2;
               #ERR_ALERT_3:
                   #statMonitoring.E5CC[5].Status := #ERR_ALERT_3;
               #ERR_PROGRAM_END_OUTPUT:
                   #statMonitoring.E5CC[5].Status := #ERR_PROGRAM_END_OUTPUT;
               #ERR_EVENT_INPUT_1:
                   #statMonitoring.E5CC[5].Status := #ERR_EVENT_INPUT_1;
               #ERR_EVENT_INPUT_2:
                   #statMonitoring.E5CC[5].Status := #ERR_EVENT_INPUT_2;
               #ERR_EVENT_INPUT_3:
                   #statMonitoring.E5CC[5].Status := #ERR_EVENT_INPUT_3;
               #ERR_EVENT_INPUT_4:
                   #statMonitoring.E5CC[5].Status := #ERR_EVENT_INPUT_4;
               #ERR_WRITE_MODE:
                   #statMonitoring.E5CC[5].Status := #ERR_WRITE_MODE;
               #ERR_NON_VOLATILE_MEMORY:
                   #statMonitoring.E5CC[5].Status := #ERR_NON_VOLATILE_MEMORY;
               #ERR_SETTING_AREA:
                   #statMonitoring.E5CC[5].Status := #ERR_SETTING_AREA;
               #ERR_AT_RUN_STOP:
                   #statMonitoring.E5CC[5].Status := #ERR_AT_RUN_STOP;
               #ERR_RUN_STOP:
                   #statMonitoring.E5CC[5].Status := #ERR_RUN_STOP;
               #ERR_COMMUNICATION_WRITE:
                   #statMonitoring.E5CC[5].Status := #ERR_COMMUNICATION_WRITE;
               #ERR_AUTO_MANUAL:
                   #statMonitoring.E5CC[5].Status := #ERR_AUTO_MANUAL;
               #ERR_PROGRAM_START:
                   #statMonitoring.E5CC[5].Status := #ERR_PROGRAM_START;
               #ERR_HEATER_CURRENT_VALUE_EXCEEDED_CT2:
                   #statMonitoring.E5CC[5].Status := #ERR_HEATER_CURRENT_VALUE_EXCEEDED_CT2;
               #ERR_HEATER_CURRENT_VALUE_HOLD_CT2:
                   #statMonitoring.E5CC[5].Status := #ERR_HEATER_CURRENT_VALUE_HOLD_CT2;
               #ERR_HS_SSR_FAILURE_ALARM_CT2:
                   #statMonitoring.E5CC[5].Status := #ERR_HS_SSR_FAILURE_ALARM_CT2;
           END_CASE;
       ELSIF #"statE5CC[5]".statReadStatus = 0 THEN
           #statMonitoring.E5CC[5].Status := 0;
       END_IF;
   END_REGION

   #statMonitoring.E5CC[5].Error := #"statE5CC[5]".statReadStatus <> 0;
END_REGION

REGION Network 81 (SCL): E5CC[5]-##### Outputs mapping #####
   // Output Mapping
   #statMonitoring.E5CC[5].Temp_SP := #"statE5CC[5]".statTempSP;
   #statMonitoring.E5CC[5].Temp_AlarmValue1 := #"statE5CC[5]".statAlarmValue1;
   #statMonitoring.E5CC[5].Temp_AlarmValue1_UpperLimit := #"statE5CC[5]".statAlarmValue1_UpperLimit;
   #statMonitoring.E5CC[5].Temp_AlarmValue1_LowerLimit := #"statE5CC[5]".statAlarmValue1_LowerLimit;
   #statMonitoring.E5CC[5].Temp_AlarmValue2 := #"statE5CC[5]".statAlarmValue2;
   #statMonitoring.E5CC[5].Temp_AlarmValue2_UpperLimit := #"statE5CC[5]".statAlarmValue2_UpperLimit;
   #statMonitoring.E5CC[5].Temp_AlarmValue2_LowerLimit := #"statE5CC[5]".statAlarmValue2_LowerLimit;
   #statMonitoring.E5CC[5].E5CC_Status := #"statE5CC[5]".statReadStatus;
   #statMonitoring.E5CC[5].E5CC_Status_Bool := #"statE5CC[5]".statReadStatus_Bool;
END_REGION

REGION Network 82 (SCL): ###### Output Mapping ######
   // Monitoring
   IF #statCurrentUnit = 1 THEN
       #statMBMasterBuffer[1].BUSY := #statConfiguration.MB_Master.BUSY;
       #statMBMasterBuffer[1].ERROR := #statConfiguration.MB_Master.ERROR;
       #statMBMasterBuffer[1].STATUS := #statConfiguration.MB_Master.STATUS;
   END_IF;
   IF #statCurrentUnit = 2 THEN
       #statMBMasterBuffer[2].BUSY := #statConfiguration.MB_Master.BUSY;
       #statMBMasterBuffer[2].ERROR := #statConfiguration.MB_Master.ERROR;
       #statMBMasterBuffer[2].STATUS := #statConfiguration.MB_Master.STATUS;
   END_IF;
   IF #statCurrentUnit = 3 THEN
       #statMBMasterBuffer[3].BUSY := #statConfiguration.MB_Master.BUSY;
       #statMBMasterBuffer[3].ERROR := #statConfiguration.MB_Master.ERROR;
       #statMBMasterBuffer[3].STATUS := #statConfiguration.MB_Master.STATUS;
   END_IF;
   IF #statCurrentUnit = 4 THEN
       #statMBMasterBuffer[4].BUSY := #statConfiguration.MB_Master.BUSY;
       #statMBMasterBuffer[4].ERROR := #statConfiguration.MB_Master.ERROR;
       #statMBMasterBuffer[4].STATUS := #statConfiguration.MB_Master.STATUS;
   END_IF;
   IF #statCurrentUnit = 5 THEN
       #statMBMasterBuffer[5].BUSY := #statConfiguration.MB_Master.BUSY;
       #statMBMasterBuffer[5].ERROR := #statConfiguration.MB_Master.ERROR;
       #statMBMasterBuffer[5].STATUS := #statConfiguration.MB_Master.STATUS;
   END_IF;
   #controlNode.monitoring.E5CC[1] := #moduleInterface.monitoring.E5CC[1] := #statMonitoring.E5CC[1];
   #controlNode.monitoring.E5CC[2] := #moduleInterface.monitoring.E5CC[2] := #statMonitoring.E5CC[2];
   #controlNode.monitoring.E5CC[3] := #moduleInterface.monitoring.E5CC[3] := #statMonitoring.E5CC[3];
   #controlNode.monitoring.E5CC[4] := #moduleInterface.monitoring.E5CC[4] := #statMonitoring.E5CC[4];
   #controlNode.monitoring.E5CC[5] := #moduleInterface.monitoring.E5CC[5] := #statMonitoring.E5CC[5];
END_REGION
END_FUNCTION_BLOCK
